SPLINE
SPL {X  -127.452, Y  +285.790, Z    +0.000, E1   +56.591, E3 +27659.937}
SPL {X  -151.591, Y  +331.344, Z    +0.000, E1   +43.870, E3 +27676.036}
SPL {X  -158.135, Y  +358.205, Z    +0.000, E1   +26.984, E3 +27679.764}
SPL {X  -159.602, Y  +371.361, Z    +0.000, E1   +14.835, E3 +27680.660}
SPL {X  -159.981, Y  +380.818, Z    +0.000, E1    +4.512, E3 +27680.938}
SPL {X  -159.990, Y  +384.681, Z    +0.000, E1    -0.222, E3 +27680.967}
SPL {X  -159.990, Y  +387.626, Z    +0.000, E1    -8.190, E3 +27680.995}
SPL {X  -159.990, Y  +390.340, Z    +0.000, E1   -15.987, E3 +27681.060}
SPL {X  -159.990, Y  +394.216, Z    +0.000, E1   -27.062, E3 +27681.222}
SPL {X  -159.990, Y  +399.855, Z    +0.000, E1   -40.916, E3 +27681.593}
SPL {X  -159.990, Y  +405.475, Z    +0.000, E1   -51.039, E3 +27682.110}
SPL {X  -159.990, Y  +414.231, Z    +0.000, E1   -60.575, E3 +27683.294}
SPL {X  -159.990, Y  +462.953, Z    +0.000, E1   -73.611, E3 +27695.033}
SPL {X  -153.839, Y  +715.436, Z    +0.000, E1   -75.884, E3 +27797.463}
SPL {X  -148.840, Y  +730.182, Z    +0.000, E1   -75.434, E3 +27810.040}
SPL {X  -143.409, Y  +742.426, Z    +0.000, E1   -74.905, E3 +27821.552}
SPL {X  -139.557, Y  +749.735, Z    +0.000, E1   -74.483, E3 +27828.900}
SPL {X  -136.371, Y  +755.165, Z    +0.000, E1   -74.152, E3 +27834.446}
SPL {X  -133.102, Y  +760.274, Z    +0.000, E1   -73.777, E3 +27839.831}
SPL {X  -128.975, Y  +766.169, Z    +0.000, E1   -73.313, E3 +27846.106}
SPL {X  -124.947, Y  +771.425, Z    +0.000, E1   -72.782, E3 +27851.799}
SPL {X  -121.698, Y  +775.357, Z    +0.000, E1   -72.353, E3 +27855.994}
SPL {X  -118.622, Y  +778.858, Z    +0.000, E1   -71.924, E3 +27859.620}
SPL {X   -66.171, Y  +817.165, Z    +0.000, E1   -56.016, E3 +28010.978}
ENDSPLINE

SPLINE
SPL {X  -126.418, Y  +769.557, Z    +0.000, E1   -57.118, E3 +28194.219}
SPL {X  -148.476, Y  +731.097, Z    +0.000, E1   -47.824, E3 +28209.375}
SPL {X  -156.642, Y  +704.059, Z    +0.000, E1   -33.659, E3 +28214.017}
SPL {X  -159.317, Y  +686.157, Z    +0.000, E1   -18.660, E3 +28215.507}
SPL {X  -159.973, Y  +673.799, Z    +0.000, E1    -5.345, E3 +28215.956}
SPL {X  -159.990, Y  +669.500, Z    +0.000, E1    +0.000, E3 +28215.996}
SPL {X  -159.990, Y  +667.794, Z    +0.000, E1    +4.255, E3 +28216.007}
SPL {X  -159.990, Y  +664.091, Z    +0.000, E1   +14.928, E3 +28216.079}
SPL {X  -159.990, Y  +659.599, Z    +0.000, E1   +28.016, E3 +28216.250}
SPL {X  -159.990, Y  +652.711, Z    +0.000, E1   +44.293, E3 +28216.729}
SPL {X  -159.990, Y  +640.730, Z    +0.000, E1   +60.297, E3 +28218.078}
SPL {X  -159.990, Y  +620.478, Z    +0.000, E1   +70.026, E3 +28221.891}
SPL {X  -159.990, Y  +573.021, Z    +0.000, E1   +74.619, E3 +28235.835}
SPL {X  -154.165, Y  +339.724, Z    +0.000, E1   +75.927, E3 +28331.682}
SPL {X  -150.223, Y  +327.456, Z    +0.000, E1   +75.573, E3 +28341.947}
SPL {X  -136.549, Y  +299.126, Z    +0.000, E1   +77.537, E3 +28334.837}
ENDSPLINE

SPLINE
SPL {X  -136.862, Y  +299.641, Z    +0.000, E1   +76.604, E3 +28343.479}
ENDSPLINE

SPLINE
SPL {X  -136.434, Y  +298.938, Z    +0.000, E1   +75.982, E3 +28349.370}
SPL {X  -135.890, Y  +298.057, Z    +0.000, E1   +75.040, E3 +28357.836}
SPL {X  -134.349, Y  +295.626, Z    +0.000, E1   +74.322, E3 +28364.683}
SPL {X  -131.287, Y  +291.064, Z    +0.000, E1   +73.972, E3 +28369.496}
SPL {X  -128.265, Y  +286.871, Z    +0.000, E1   +73.613, E3 +28373.952}
SPL {X  -125.161, Y  +282.843, Z    +0.000, E1   +73.232, E3 +28378.224}
SPL {X  -122.038, Y  +279.042, Z    +0.000, E1   +72.832, E3 +28382.204}
SPL {X  -118.642, Y  +275.165, Z    +0.000, E1   +72.381, E3 +28386.167}
SPL {X   -66.040, Y  +236.776, Z    +0.000, E1   +55.694, E3 +28547.530}
ENDSPLINE

SPLINE
SPL {X  -127.452, Y  +285.790, Z    +0.000, E1   +56.591, E3 +28721.476}
SPL {X  -151.591, Y  +331.344, Z    +0.000, E1   +43.870, E3 +28737.575}
SPL {X  -158.135, Y  +358.205, Z    +0.000, E1   +26.984, E3 +28741.302}
SPL {X  -159.602, Y  +371.361, Z    +0.000, E1   +14.835, E3 +28742.198}
SPL {X  -159.981, Y  +380.818, Z    +0.000, E1    +4.512, E3 +28742.476}
SPL {X  -159.990, Y  +384.681, Z    +0.000, E1    -0.222, E3 +28742.505}
SPL {X  -159.990, Y  +387.626, Z    +0.000, E1    -8.190, E3 +28742.534}
SPL {X  -159.990, Y  +390.340, Z    +0.000, E1   -15.987, E3 +28742.598}
SPL {X  -159.990, Y  +394.216, Z    +0.000, E1   -27.062, E3 +28742.760}
SPL {X  -159.990, Y  +399.855, Z    +0.000, E1   -40.916, E3 +28743.131}
SPL {X  -159.990, Y  +405.475, Z    +0.000, E1   -51.039, E3 +28743.648}
SPL {X  -159.990, Y  +414.231, Z    +0.000, E1   -60.575, E3 +28744.832}
SPL {X  -159.990, Y  +462.953, Z    +0.000, E1   -73.611, E3 +28756.571}
SPL {X  -153.839, Y  +715.436, Z    +0.000, E1   -75.884, E3 +28859.002}
SPL {X  -148.840, Y  +730.182, Z    +0.000, E1   -75.434, E3 +28871.578}
SPL {X  -143.409, Y  +742.426, Z    +0.000, E1   -74.905, E3 +28883.090}
SPL {X  -139.557, Y  +749.735, Z    +0.000, E1   -74.483, E3 +28890.439}
SPL {X  -136.371, Y  +755.165, Z    +0.000, E1   -74.152, E3 +28895.984}
SPL {X  -133.102, Y  +760.274, Z    +0.000, E1   -73.777, E3 +28901.369}
SPL {X  -128.975, Y  +766.169, Z    +0.000, E1   -73.313, E3 +28907.645}
SPL {X  -124.947, Y  +771.425, Z    +0.000, E1   -72.782, E3 +28913.338}
SPL {X  -121.698, Y  +775.357, Z    +0.000, E1   -72.353, E3 +28917.532}
SPL {X  -118.622, Y  +778.858, Z    +0.000, E1   -71.924, E3 +28921.158}
SPL {X   -66.171, Y  +817.165, Z    +0.000, E1   -56.016, E3 +29072.517}
ENDSPLINE

SPLINE
SPL {X  -126.418, Y  +769.557, Z    +0.000, E1   -57.118, E3 +29255.758}
SPL {X  -148.476, Y  +731.097, Z    +0.000, E1   -47.824, E3 +29270.914}
SPL {X  -156.642, Y  +704.059, Z    +0.000, E1   -33.659, E3 +29275.555}
SPL {X  -159.317, Y  +686.157, Z    +0.000, E1   -18.660, E3 +29277.046}
SPL {X  -159.973, Y  +673.799, Z    +0.000, E1    -5.345, E3 +29277.494}
SPL {X  -159.990, Y  +669.500, Z    +0.000, E1    +0.000, E3 +29277.534}
SPL {X  -159.990, Y  +667.794, Z    +0.000, E1    +4.255, E3 +29277.546}
SPL {X  -159.990, Y  +664.091, Z    +0.000, E1   +14.928, E3 +29277.618}
SPL {X  -159.990, Y  +659.599, Z    +0.000, E1   +28.016, E3 +29277.788}
SPL {X  -159.990, Y  +652.711, Z    +0.000, E1   +44.293, E3 +29278.268}
SPL {X  -159.990, Y  +640.730, Z    +0.000, E1   +60.297, E3 +29279.617}
SPL {X  -159.990, Y  +620.478, Z    +0.000, E1   +70.026, E3 +29283.430}
SPL {X  -159.990, Y  +573.021, Z    +0.000, E1   +74.619, E3 +29297.374}
SPL {X  -154.165, Y  +339.724, Z    +0.000, E1   +75.927, E3 +29393.221}
SPL {X  -150.223, Y  +327.456, Z    +0.000, E1   +75.573, E3 +29403.486}
SPL {X  -136.549, Y  +299.126, Z    +0.000, E1   +77.537, E3 +29396.376}
ENDSPLINE

SPLINE
SPL {X  -136.862, Y  +299.641, Z    +0.000, E1   +76.604, E3 +29405.018}
ENDSPLINE

SPLINE
SPL {X  -136.434, Y  +298.938, Z    +0.000, E1   +75.982, E3 +29410.909}
SPL {X  -135.890, Y  +298.057, Z    +0.000, E1   +75.040, E3 +29419.375}
SPL {X  -134.349, Y  +295.626, Z    +0.000, E1   +74.322, E3 +29426.222}
SPL {X  -131.287, Y  +291.064, Z    +0.000, E1   +73.972, E3 +29431.034}
SPL {X  -128.265, Y  +286.871, Z    +0.000, E1   +73.613, E3 +29435.490}
SPL {X  -125.161, Y  +282.843, Z    +0.000, E1   +73.232, E3 +29439.762}
SPL {X  -122.038, Y  +279.042, Z    +0.000, E1   +72.832, E3 +29443.742}
SPL {X  -118.642, Y  +275.165, Z    +0.000, E1   +72.381, E3 +29447.705}
SPL {X   -66.040, Y  +236.776, Z    +0.000, E1   +55.694, E3 +29609.069}
ENDSPLINE

SPLINE
SPL {X  -127.452, Y  +285.790, Z    +0.000, E1   +56.591, E3 +29783.014}
SPL {X  -151.591, Y  +331.344, Z    +0.000, E1   +43.870, E3 +29799.113}
SPL {X  -158.135, Y  +358.205, Z    +0.000, E1   +26.984, E3 +29802.841}
SPL {X  -159.602, Y  +371.361, Z    +0.000, E1   +14.835, E3 +29803.737}
SPL {X  -159.981, Y  +380.818, Z    +0.000, E1    +4.512, E3 +29804.015}
SPL {X  -159.990, Y  +384.681, Z    +0.000, E1    -0.222, E3 +29804.044}
SPL {X  -159.990, Y  +387.626, Z    +0.000, E1    -8.190, E3 +29804.072}
SPL {X  -159.990, Y  +390.340, Z    +0.000, E1   -15.987, E3 +29804.137}
SPL {X  -159.990, Y  +394.216, Z    +0.000, E1   -27.062, E3 +29804.299}
SPL {X  -159.990, Y  +399.855, Z    +0.000, E1   -40.916, E3 +29804.670}
SPL {X  -159.990, Y  +405.475, Z    +0.000, E1   -51.039, E3 +29805.187}
SPL {X  -159.990, Y  +414.231, Z    +0.000, E1   -60.575, E3 +29806.371}
SPL {X  -159.990, Y  +462.953, Z    +0.000, E1   -73.611, E3 +29818.110}
SPL {X  -153.839, Y  +715.436, Z    +0.000, E1   -75.884, E3 +29920.540}
SPL {X  -149.923, Y  +727.355, Z    +0.000, E1   -75.515, E3 +29930.650}
SPL {X  -145.995, Y  +736.939, Z    +0.000, E1   -75.150, E3 +29939.385}
SPL {X  -141.012, Y  +747.080, Z    +0.000, E1   -74.661, E3 +29949.237}
SPL {X  -136.371, Y  +755.165, Z    +0.000, E1   -74.152, E3 +29957.523}
SPL {X  -133.102, Y  +760.274, Z    +0.000, E1   -73.777, E3 +29962.908}
SPL {X  -128.975, Y  +766.169, Z    +0.000, E1   -73.313, E3 +29969.183}
SPL {X  -124.947, Y  +771.425, Z    +0.000, E1   -72.782, E3 +29974.876}
SPL {X  -121.698, Y  +775.357, Z    +0.000, E1   -72.353, E3 +29979.071}
SPL {X  -118.622, Y  +778.858, Z    +0.000, E1   -71.924, E3 +29982.697}
SPL {X   -66.171, Y  +817.165, Z    +0.000, E1   -56.016, E3 +30134.055}
ENDSPLINE

SPLINE
SPL {X  -126.418, Y  +769.557, Z    +0.000, E1   -57.118, E3 +30317.296}
SPL {X  -148.476, Y  +731.097, Z    +0.000, E1   -47.824, E3 +30332.452}
SPL {X  -156.642, Y  +704.059, Z    +0.000, E1   -33.659, E3 +30337.094}
SPL {X  -159.317, Y  +686.157, Z    +0.000, E1   -18.660, E3 +30338.584}
SPL {X  -159.907, Y  +676.666, Z    +0.000, E1    -8.555, E3 +30338.982}
SPL {X  -159.990, Y  +669.586, Z    +0.000, E1    -0.216, E3 +30339.073}
SPL {X  -159.990, Y  +667.794, Z    +0.000, E1    +4.255, E3 +30339.084}
SPL {X  -159.990, Y  +664.091, Z    +0.000, E1   +14.928, E3 +30339.156}
SPL {X  -159.990, Y  +659.599, Z    +0.000, E1   +28.016, E3 +30339.327}
SPL {X  -159.990, Y  +652.711, Z    +0.000, E1   +44.293, E3 +30339.806}
SPL {X  -159.990, Y  +640.730, Z    +0.000, E1   +60.297, E3 +30341.155}
SPL {X  -159.990, Y  +620.478, Z    +0.000, E1   +70.026, E3 +30344.968}
SPL {X  -159.990, Y  +573.021, Z    +0.000, E1   +74.619, E3 +30358.912}
SPL {X  -154.165, Y  +339.724, Z    +0.000, E1   +75.927, E3 +30454.759}
SPL {X  -150.223, Y  +327.456, Z    +0.000, E1   +75.573, E3 +30465.024}
SPL {X  -136.549, Y  +299.126, Z    +0.000, E1   +77.537, E3 +30457.914}
ENDSPLINE

SPLINE
SPL {X  -136.862, Y  +299.641, Z    +0.000, E1   +76.604, E3 +30466.556}
ENDSPLINE

SPLINE
SPL {X  -136.434, Y  +298.938, Z    +0.000, E1   +75.982, E3 +30472.447}
SPL {X  -135.890, Y  +298.057, Z    +0.000, E1   +75.040, E3 +30480.913}
SPL {X  -134.349, Y  +295.626, Z    +0.000, E1   +74.322, E3 +30487.760}
SPL {X  -131.287, Y  +291.064, Z    +0.000, E1   +73.972, E3 +30492.573}
SPL {X  -128.265, Y  +286.871, Z    +0.000, E1   +73.613, E3 +30497.029}
SPL {X  -125.161, Y  +282.843, Z    +0.000, E1   +73.232, E3 +30501.301}
SPL {X  -122.038, Y  +279.042, Z    +0.000, E1   +72.832, E3 +30505.281}
SPL {X  -118.642, Y  +275.165, Z    +0.000, E1   +72.381, E3 +30509.244}
SPL {X   -66.040, Y  +236.776, Z    +0.000, E1   +55.694, E3 +30670.607}
ENDSPLINE

SPLINE
SPL {X  -127.452, Y  +285.790, Z    +0.000, E1   +56.591, E3 +30844.552}
SPL {X  -148.001, Y  +321.733, Z    +0.000, E1   +47.810, E3 +30858.656}
SPL {X  -154.604, Y  +341.337, Z    +0.000, E1   +38.630, E3 +30862.430}
SPL {X  -158.135, Y  +358.205, Z    +0.000, E1   +26.984, E3 +30864.379}
SPL {X  -159.602, Y  +371.361, Z    +0.000, E1   +14.835, E3 +30865.275}
SPL {X  -159.981, Y  +380.818, Z    +0.000, E1    +4.512, E3 +30865.553}
SPL {X  -159.990, Y  +384.681, Z    +0.000, E1    -0.222, E3 +30865.582}
SPL {X  -159.990, Y  +389.079, Z    +0.000, E1   -12.017, E3 +30865.645}
SPL {X  -159.990, Y  +394.216, Z    +0.000, E1   -27.062, E3 +30865.837}
SPL {X  -159.990, Y  +399.855, Z    +0.000, E1   -40.916, E3 +30866.208}
SPL {X  -159.990, Y  +405.475, Z    +0.000, E1   -51.039, E3 +30866.725}
SPL {X  -159.990, Y  +414.231, Z    +0.000, E1   -60.575, E3 +30867.909}
SPL {X  -159.990, Y  +462.953, Z    +0.000, E1   -73.611, E3 +30879.648}
SPL {X  -153.839, Y  +715.436, Z    +0.000, E1   -75.884, E3 +30982.079}
SPL {X  -148.840, Y  +730.182, Z    +0.000, E1   -75.434, E3 +30994.655}
SPL {X  -143.409, Y  +742.426, Z    +0.000, E1   -74.905, E3 +31006.167}
SPL {X  -139.557, Y  +749.735, Z    +0.000, E1   -74.483, E3 +31013.515}
SPL {X  -136.371, Y  +755.165, Z    +0.000, E1   -74.152, E3 +31019.061}
SPL {X  -133.102, Y  +760.274, Z    +0.000, E1   -73.777, E3 +31024.446}
SPL {X  -128.975, Y  +766.169, Z    +0.000, E1   -73.313, E3 +31030.722}
SPL {X  -124.947, Y  +771.425, Z    +0.000, E1   -72.782, E3 +31036.415}
SPL {X  -121.698, Y  +775.357, Z    +0.000, E1   -72.353, E3 +31040.609}
SPL {X  -118.622, Y  +778.858, Z    +0.000, E1   -71.924, E3 +31044.235}
SPL {X   -66.171, Y  +817.165, Z    +0.000, E1   -56.016, E3 +31195.593}
ENDSPLINE

SPLINE
SPL {X  -126.418, Y  +769.557, Z    +0.000, E1   -57.118, E3 +31378.835}
SPL {X  -145.244, Y  +738.589, Z    +0.000, E1   -50.405, E3 +31392.076}
SPL {X  -150.151, Y  +726.741, Z    +0.000, E1   -46.068, E3 +31395.003}
SPL {X  -156.642, Y  +704.059, Z    +0.000, E1   -33.659, E3 +31398.632}
SPL {X  -159.317, Y  +686.157, Z    +0.000, E1   -18.660, E3 +31400.123}
SPL {X  -159.973, Y  +673.799, Z    +0.000, E1    -5.345, E3 +31400.571}
SPL {X  -159.990, Y  +669.500, Z    +0.000, E1    +0.000, E3 +31400.611}
SPL {X  -159.990, Y  +667.794, Z    +0.000, E1    +4.255, E3 +31400.623}
SPL {X  -159.990, Y  +664.091, Z    +0.000, E1   +14.928, E3 +31400.695}
SPL {X  -159.990, Y  +658.301, Z    +0.000, E1   +31.283, E3 +31400.947}
SPL {X  -159.990, Y  +650.845, Z    +0.000, E1   +47.892, E3 +31401.492}
SPL {X  -159.990, Y  +640.730, Z    +0.000, E1   +60.297, E3 +31402.693}
SPL {X  -159.990, Y  +620.478, Z    +0.000, E1   +70.026, E3 +31406.507}
SPL {X  -159.990, Y  +573.021, Z    +0.000, E1   +74.619, E3 +31420.451}
SPL {X  -154.165, Y  +339.724, Z    +0.000, E1   +75.927, E3 +31516.298}
SPL {X  -150.223, Y  +327.456, Z    +0.000, E1   +75.573, E3 +31526.562}
SPL {X  -136.549, Y  +299.126, Z    +0.000, E1   +77.537, E3 +31519.452}
ENDSPLINE

SPLINE
SPL {X  -136.862, Y  +299.641, Z    +0.000, E1   +76.604, E3 +31528.094}
ENDSPLINE

SPLINE
SPL {X  -136.434, Y  +298.938, Z    +0.000, E1   +75.982, E3 +31533.986}
SPL {X  -135.890, Y  +298.057, Z    +0.000, E1   +75.040, E3 +31542.452}
SPL {X  -134.349, Y  +295.626, Z    +0.000, E1   +74.322, E3 +31549.299}
SPL {X  -131.287, Y  +291.064, Z    +0.000, E1   +73.972, E3 +31554.111}
SPL {X  -128.265, Y  +286.871, Z    +0.000, E1   +73.613, E3 +31558.567}
SPL {X  -125.161, Y  +282.843, Z    +0.000, E1   +73.232, E3 +31562.839}
SPL {X  -122.038, Y  +279.042, Z    +0.000, E1   +72.832, E3 +31566.819}
SPL {X  -118.642, Y  +275.165, Z    +0.000, E1   +72.381, E3 +31570.782}
SPL {X   -66.040, Y  +236.776, Z    +0.000, E1   +55.694, E3 +31732.146}
ENDSPLINE

SPLINE
SPL {X  -127.452, Y  +285.790, Z    +0.000, E1   +56.591, E3 +31906.091}
SPL {X  -151.591, Y  +331.344, Z    +0.000, E1   +43.870, E3 +31922.190}
SPL {X  -158.135, Y  +358.205, Z    +0.000, E1   +26.984, E3 +31925.918}
SPL {X  -159.602, Y  +371.361, Z    +0.000, E1   +14.835, E3 +31926.814}
SPL {X  -159.981, Y  +380.818, Z    +0.000, E1    +4.512, E3 +31927.092}
SPL {X  -159.990, Y  +384.681, Z    +0.000, E1    -0.222, E3 +31927.121}
SPL {X  -159.990, Y  +387.626, Z    +0.000, E1    -8.190, E3 +31927.149}
SPL {X  -159.990, Y  +390.340, Z    +0.000, E1   -15.987, E3 +31927.214}
SPL {X  -159.990, Y  +394.216, Z    +0.000, E1   -27.062, E3 +31927.375}
SPL {X  -159.990, Y  +399.855, Z    +0.000, E1   -40.916, E3 +31927.747}
SPL {X  -159.990, Y  +405.475, Z    +0.000, E1   -51.039, E3 +31928.263}
SPL {X  -159.990, Y  +414.231, Z    +0.000, E1   -60.575, E3 +31929.448}
SPL {X  -159.990, Y  +462.953, Z    +0.000, E1   -73.611, E3 +31941.187}
SPL {X  -153.839, Y  +715.436, Z    +0.000, E1   -75.884, E3 +32043.617}
SPL {X  -149.923, Y  +727.355, Z    +0.000, E1   -75.515, E3 +32053.727}
SPL {X  -145.995, Y  +736.939, Z    +0.000, E1   -75.150, E3 +32062.462}
SPL {X  -141.012, Y  +747.080, Z    +0.000, E1   -74.661, E3 +32072.314}
SPL {X  -136.371, Y  +755.165, Z    +0.000, E1   -74.152, E3 +32080.600}
SPL {X  -131.455, Y  +762.694, Z    +0.000, E1   -73.615, E3 +32088.518}
SPL {X  -125.933, Y  +770.180, Z    +0.000, E1   -72.934, E3 +32096.582}
SPL {X  -121.698, Y  +775.357, Z    +0.000, E1   -72.353, E3 +32102.148}
SPL {X  -118.622, Y  +778.858, Z    +0.000, E1   -71.924, E3 +32105.774}
SPL {X   -66.171, Y  +817.165, Z    +0.000, E1   -56.016, E3 +32257.132}
ENDSPLINE

SPLINE
SPL {X  -126.418, Y  +769.557, Z    +0.000, E1   -57.118, E3 +32440.373}
SPL {X  -145.244, Y  +738.589, Z    +0.000, E1   -50.405, E3 +32453.615}
SPL {X  -150.151, Y  +726.741, Z    +0.000, E1   -46.068, E3 +32456.541}
SPL {X  -156.642, Y  +704.059, Z    +0.000, E1   -33.659, E3 +32460.171}
SPL {X  -159.317, Y  +686.157, Z    +0.000, E1   -18.660, E3 +32461.661}
SPL {X  -159.973, Y  +673.799, Z    +0.000, E1    -5.345, E3 +32462.110}
SPL {X  -159.990, Y  +669.500, Z    +0.000, E1    +0.000, E3 +32462.150}
SPL {X  -159.990, Y  +667.794, Z    +0.000, E1    +4.255, E3 +32462.161}
SPL {X  -159.990, Y  +664.091, Z    +0.000, E1   +14.928, E3 +32462.233}
SPL {X  -159.990, Y  +658.301, Z    +0.000, E1   +31.283, E3 +32462.486}
SPL {X  -159.990, Y  +650.845, Z    +0.000, E1   +47.892, E3 +32463.031}
SPL {X  -159.990, Y  +640.730, Z    +0.000, E1   +60.297, E3 +32464.232}
SPL {X  -159.990, Y  +620.478, Z    +0.000, E1   +70.026, E3 +32468.045}
SPL {X  -159.990, Y  +573.021, Z    +0.000, E1   +74.619, E3 +32481.989}
SPL {X  -154.165, Y  +339.724, Z    +0.000, E1   +75.927, E3 +32577.836}
SPL {X  -150.223, Y  +327.456, Z    +0.000, E1   +75.573, E3 +32588.101}
SPL {X  -136.549, Y  +299.126, Z    +0.000, E1   +77.537, E3 +32580.991}
ENDSPLINE

SPLINE
SPL {X  -136.862, Y  +299.641, Z    +0.000, E1   +76.604, E3 +32589.633}
ENDSPLINE

SPLINE
SPL {X  -136.434, Y  +298.938, Z    +0.000, E1   +75.982, E3 +32595.524}
SPL {X  -135.890, Y  +298.057, Z    +0.000, E1   +75.040, E3 +32603.990}
SPL {X  -134.349, Y  +295.626, Z    +0.000, E1   +74.322, E3 +32610.837}
SPL {X  -131.287, Y  +291.064, Z    +0.000, E1   +73.972, E3 +32615.650}
SPL {X  -128.265, Y  +286.871, Z    +0.000, E1   +73.613, E3 +32620.106}
SPL {X  -125.161, Y  +282.843, Z    +0.000, E1   +73.232, E3 +32624.378}
SPL {X  -122.038, Y  +279.042, Z    +0.000, E1   +72.832, E3 +32628.357}
SPL {X  -118.642, Y  +275.165, Z    +0.000, E1   +72.381, E3 +32632.321}
SPL {X   -66.040, Y  +236.776, Z    +0.000, E1   +55.694, E3 +32793.684}
ENDSPLINE

SPLINE
SPL {X  -127.452, Y  +285.790, Z    +0.000, E1   +56.591, E3 +32967.629}
SPL {X  -151.591, Y  +331.344, Z    +0.000, E1   +43.870, E3 +32983.729}
SPL {X  -158.135, Y  +358.205, Z    +0.000, E1   +26.984, E3 +32987.456}
SPL {X  -159.602, Y  +371.361, Z    +0.000, E1   +14.835, E3 +32988.352}
SPL {X  -159.981, Y  +380.818, Z    +0.000, E1    +4.512, E3 +32988.630}
SPL {X  -159.990, Y  +384.681, Z    +0.000, E1    -0.222, E3 +32988.659}
SPL {X  -159.990, Y  +387.626, Z    +0.000, E1    -8.190, E3 +32988.687}
SPL {X  -159.990, Y  +390.340, Z    +0.000, E1   -15.987, E3 +32988.752}
SPL {X  -159.990, Y  +394.216, Z    +0.000, E1   -27.062, E3 +32988.914}
SPL {X  -159.990, Y  +399.855, Z    +0.000, E1   -40.916, E3 +32989.285}
SPL {X  -159.990, Y  +405.475, Z    +0.000, E1   -51.039, E3 +32989.802}
SPL {X  -159.990, Y  +414.231, Z    +0.000, E1   -60.575, E3 +32990.986}
SPL {X  -159.990, Y  +462.953, Z    +0.000, E1   -73.611, E3 +33002.725}
SPL {X  -153.839, Y  +715.436, Z    +0.000, E1   -75.884, E3 +33105.156}
SPL {X  -148.840, Y  +730.182, Z    +0.000, E1   -75.434, E3 +33117.732}
SPL {X  -143.409, Y  +742.426, Z    +0.000, E1   -74.905, E3 +33129.244}
SPL {X  -139.557, Y  +749.735, Z    +0.000, E1   -74.483, E3 +33136.592}
SPL {X  -136.371, Y  +755.165, Z    +0.000, E1   -74.152, E3 +33142.138}
SPL {X  -133.102, Y  +760.274, Z    +0.000, E1   -73.777, E3 +33147.523}
SPL {X  -128.975, Y  +766.169, Z    +0.000, E1   -73.313, E3 +33153.799}
SPL {X  -124.947, Y  +771.425, Z    +0.000, E1   -72.782, E3 +33159.492}
SPL {X  -121.698, Y  +775.357, Z    +0.000, E1   -72.353, E3 +33163.686}
SPL {X  -118.622, Y  +778.858, Z    +0.000, E1   -71.924, E3 +33167.312}
SPL {X   -66.171, Y  +817.165, Z    +0.000, E1   -56.016, E3 +33318.670}
ENDSPLINE

SPLINE
SPL {X  -126.418, Y  +769.557, Z    +0.000, E1   -57.118, E3 +33501.912}
SPL {X  -145.244, Y  +738.589, Z    +0.000, E1   -50.405, E3 +33515.153}
SPL {X  -150.151, Y  +726.741, Z    +0.000, E1   -46.068, E3 +33518.080}
SPL {X  -156.642, Y  +704.059, Z    +0.000, E1   -33.659, E3 +33521.709}
SPL {X  -159.317, Y  +686.157, Z    +0.000, E1   -18.660, E3 +33523.200}
SPL {X  -159.973, Y  +673.799, Z    +0.000, E1    -5.345, E3 +33523.648}
SPL {X  -159.990, Y  +669.500, Z    +0.000, E1    +0.000, E3 +33523.688}
SPL {X  -159.990, Y  +667.794, Z    +0.000, E1    +4.255, E3 +33523.699}
SPL {X  -159.990, Y  +664.091, Z    +0.000, E1   +14.928, E3 +33523.772}
SPL {X  -159.990, Y  +659.599, Z    +0.000, E1   +28.016, E3 +33523.942}
SPL {X  -159.990, Y  +652.711, Z    +0.000, E1   +44.293, E3 +33524.421}
SPL {X  -159.990, Y  +640.730, Z    +0.000, E1   +60.297, E3 +33525.770}
SPL {X  -159.990, Y  +620.478, Z    +0.000, E1   +70.026, E3 +33529.584}
SPL {X  -159.990, Y  +573.021, Z    +0.000, E1   +74.619, E3 +33543.528}
SPL {X  -154.165, Y  +339.724, Z    +0.000, E1   +75.927, E3 +33639.374}
SPL {X  -150.571, Y  +328.416, Z    +0.000, E1   +75.599, E3 +33648.820}
SPL {X  -148.206, Y  +322.236, Z    +0.000, E1   +75.365, E3 +33654.364}
SPL {X  -136.549, Y  +299.126, Z    +0.000, E1   +77.537, E3 +33642.529}
ENDSPLINE

SPLINE
SPL {X  -136.862, Y  +299.641, Z    +0.000, E1   +76.604, E3 +33651.171}
ENDSPLINE

SPLINE
SPL {X  -136.434, Y  +298.938, Z    +0.000, E1   +75.982, E3 +33657.062}
SPL {X  -135.890, Y  +298.057, Z    +0.000, E1   +75.040, E3 +33665.528}
SPL {X  -134.349, Y  +295.626, Z    +0.000, E1   +74.322, E3 +33672.376}
SPL {X  -131.287, Y  +291.064, Z    +0.000, E1   +73.972, E3 +33677.188}
SPL {X  -128.265, Y  +286.871, Z    +0.000, E1   +73.613, E3 +33681.644}
SPL {X  -125.161, Y  +282.843, Z    +0.000, E1   +73.232, E3 +33685.916}
SPL {X  -122.038, Y  +279.042, Z    +0.000, E1   +72.832, E3 +33689.896}
SPL {X  -118.642, Y  +275.165, Z    +0.000, E1   +72.381, E3 +33693.859}
SPL {X   -66.040, Y  +236.776, Z    +0.000, E1   +55.694, E3 +33855.223}
ENDSPLINE

SPLINE
SPL {X  -127.452, Y  +285.790, Z    +0.000, E1   +56.591, E3 +34029.168}
SPL {X  -151.591, Y  +331.344, Z    +0.000, E1   +43.870, E3 +34045.267}
SPL {X  -158.135, Y  +358.205, Z    +0.000, E1   +26.984, E3 +34048.995}
SPL {X  -159.602, Y  +371.361, Z    +0.000, E1   +14.835, E3 +34049.891}
SPL {X  -159.981, Y  +380.818, Z    +0.000, E1    +4.512, E3 +34050.169}
SPL {X  -159.990, Y  +384.681, Z    +0.000, E1    -0.222, E3 +34050.198}
SPL {X  -159.990, Y  +387.626, Z    +0.000, E1    -8.190, E3 +34050.226}
SPL {X  -159.990, Y  +390.340, Z    +0.000, E1   -15.987, E3 +34050.290}
SPL {X  -159.990, Y  +394.216, Z    +0.000, E1   -27.062, E3 +34050.452}
SPL {X  -159.990, Y  +399.855, Z    +0.000, E1   -40.916, E3 +34050.823}
SPL {X  -159.990, Y  +405.475, Z    +0.000, E1   -51.039, E3 +34051.340}
SPL {X  -159.990, Y  +414.231, Z    +0.000, E1   -60.575, E3 +34052.525}
SPL {X  -159.990, Y  +462.953, Z    +0.000, E1   -73.611, E3 +34064.264}
SPL {X  -153.839, Y  +715.436, Z    +0.000, E1   -75.884, E3 +34166.694}
SPL {X  -148.840, Y  +730.182, Z    +0.000, E1   -75.434, E3 +34179.271}
SPL {X  -143.409, Y  +742.426, Z    +0.000, E1   -74.905, E3 +34190.783}
SPL {X  -139.557, Y  +749.735, Z    +0.000, E1   -74.483, E3 +34198.131}
SPL {X  -136.371, Y  +755.165, Z    +0.000, E1   -74.152, E3 +34203.677}
SPL {X  -133.102, Y  +760.274, Z    +0.000, E1   -73.777, E3 +34209.062}
SPL {X  -128.975, Y  +766.169, Z    +0.000, E1   -73.313, E3 +34215.337}
SPL {X  -124.947, Y  +771.425, Z    +0.000, E1   -72.782, E3 +34221.030}
SPL {X  -121.698, Y  +775.357, Z    +0.000, E1   -72.353, E3 +34225.225}
SPL {X  -118.622, Y  +778.858, Z    +0.000, E1   -71.924, E3 +34228.851}
SPL {X   -66.171, Y  +817.165, Z    +0.000, E1   -56.016, E3 +34380.209}
ENDSPLINE

SPLINE
SPL {X  -126.418, Y  +769.557, Z    +0.000, E1   -57.118, E3 +34563.450}
SPL {X  -148.476, Y  +731.097, Z    +0.000, E1   -47.824, E3 +34578.606}
SPL {X  -156.642, Y  +704.059, Z    +0.000, E1   -33.659, E3 +34583.248}
SPL {X  -159.317, Y  +686.157, Z    +0.000, E1   -18.660, E3 +34584.738}
SPL {X  -159.973, Y  +673.799, Z    +0.000, E1    -5.345, E3 +34585.187}
SPL {X  -159.990, Y  +669.500, Z    +0.000, E1    +0.000, E3 +34585.227}
SPL {X  -159.990, Y  +667.794, Z    +0.000, E1    +4.255, E3 +34585.238}
SPL {X  -159.990, Y  +664.091, Z    +0.000, E1   +14.928, E3 +34585.310}
SPL {X  -159.990, Y  +659.599, Z    +0.000, E1   +28.016, E3 +34585.480}
SPL {X  -159.990, Y  +652.711, Z    +0.000, E1   +44.293, E3 +34585.960}
SPL {X  -159.990, Y  +640.730, Z    +0.000, E1   +60.297, E3 +34587.309}
SPL {X  -159.990, Y  +620.478, Z    +0.000, E1   +70.026, E3 +34591.122}
SPL {X  -159.990, Y  +573.021, Z    +0.000, E1   +74.619, E3 +34605.066}
SPL {X  -154.165, Y  +339.724, Z    +0.000, E1   +75.927, E3 +34700.913}
SPL {X  -150.223, Y  +327.456, Z    +0.000, E1   +75.573, E3 +34711.178}
SPL {X  -136.549, Y  +299.126, Z    +0.000, E1   +77.537, E3 +34704.068}
ENDSPLINE

SPLINE
SPL {X  -136.862, Y  +299.641, Z    +0.000, E1   +76.604, E3 +34712.710}
ENDSPLINE

SPLINE
SPL {X  -136.434, Y  +298.938, Z    +0.000, E1   +75.982, E3 +34718.601}
SPL {X  -135.890, Y  +298.057, Z    +0.000, E1   +75.040, E3 +34727.067}
SPL {X  -134.349, Y  +295.626, Z    +0.000, E1   +74.322, E3 +34733.914}
SPL {X  -131.287, Y  +291.064, Z    +0.000, E1   +73.972, E3 +34738.727}
SPL {X  -128.265, Y  +286.871, Z    +0.000, E1   +73.613, E3 +34743.183}
SPL {X  -125.161, Y  +282.843, Z    +0.000, E1   +73.232, E3 +34747.454}
SPL {X  -122.038, Y  +279.042, Z    +0.000, E1   +72.832, E3 +34751.434}
SPL {X  -118.642, Y  +275.165, Z    +0.000, E1   +72.381, E3 +34755.398}
SPL {X   -66.040, Y  +236.776, Z    +0.000, E1   +55.694, E3 +34916.761}
ENDSPLINE

SPLINE
SPL {X  -127.452, Y  +285.790, Z    +0.000, E1   +56.591, E3 +35090.706}
SPL {X  -151.591, Y  +331.344, Z    +0.000, E1   +43.870, E3 +35106.806}
SPL {X  -158.135, Y  +358.205, Z    +0.000, E1   +26.984, E3 +35110.533}
SPL {X  -159.602, Y  +371.361, Z    +0.000, E1   +14.835, E3 +35111.429}
SPL {X  -159.981, Y  +380.818, Z    +0.000, E1    +4.512, E3 +35111.707}
SPL {X  -159.990, Y  +384.681, Z    +0.000, E1    -0.222, E3 +35111.736}
SPL {X  -159.990, Y  +387.626, Z    +0.000, E1    -8.190, E3 +35111.764}
SPL {X  -159.990, Y  +390.340, Z    +0.000, E1   -15.987, E3 +35111.829}
SPL {X  -159.990, Y  +394.216, Z    +0.000, E1   -27.062, E3 +35111.991}
SPL {X  -159.990, Y  +399.855, Z    +0.000, E1   -40.916, E3 +35112.362}
SPL {X  -159.990, Y  +405.475, Z    +0.000, E1   -51.039, E3 +35112.879}
SPL {X  -159.990, Y  +414.231, Z    +0.000, E1   -60.575, E3 +35114.063}
SPL {X  -159.990, Y  +462.953, Z    +0.000, E1   -73.611, E3 +35125.802}
SPL {X  -153.839, Y  +715.436, Z    +0.000, E1   -75.884, E3 +35228.233}
SPL {X  -148.840, Y  +730.182, Z    +0.000, E1   -75.434, E3 +35240.809}
SPL {X  -143.409, Y  +742.426, Z    +0.000, E1   -74.905, E3 +35252.321}
SPL {X  -139.557, Y  +749.735, Z    +0.000, E1   -74.483, E3 +35259.669}
SPL {X  -136.371, Y  +755.165, Z    +0.000, E1   -74.152, E3 +35265.215}
SPL {X  -133.102, Y  +760.274, Z    +0.000, E1   -73.777, E3 +35270.600}
SPL {X  -128.975, Y  +766.169, Z    +0.000, E1   -73.313, E3 +35276.875}
SPL {X  -124.947, Y  +771.425, Z    +0.000, E1   -72.782, E3 +35282.568}
SPL {X  -121.698, Y  +775.357, Z    +0.000, E1   -72.353, E3 +35286.763}
SPL {X  -118.622, Y  +778.858, Z    +0.000, E1   -71.924, E3 +35290.389}
SPL {X   -66.171, Y  +817.165, Z    +0.000, E1   -56.016, E3 +35441.747}
ENDSPLINE

SPLINE
SPL {X  -126.418, Y  +769.557, Z    +0.000, E1   -57.118, E3 +35624.989}
SPL {X  -148.476, Y  +731.097, Z    +0.000, E1   -47.824, E3 +35640.145}
SPL {X  -156.642, Y  +704.059, Z    +0.000, E1   -33.659, E3 +35644.786}
SPL {X  -159.317, Y  +686.157, Z    +0.000, E1   -18.660, E3 +35646.276}
SPL {X  -159.973, Y  +673.799, Z    +0.000, E1    -5.345, E3 +35646.725}
SPL {X  -159.990, Y  +669.500, Z    +0.000, E1    +0.000, E3 +35646.765}
SPL {X  -159.990, Y  +667.794, Z    +0.000, E1    +4.255, E3 +35646.776}
SPL {X  -159.990, Y  +664.091, Z    +0.000, E1   +14.928, E3 +35646.848}
SPL {X  -159.990, Y  +659.599, Z    +0.000, E1   +28.016, E3 +35647.019}
SPL {X  -159.990, Y  +652.711, Z    +0.000, E1   +44.293, E3 +35647.498}
SPL {X  -159.990, Y  +640.730, Z    +0.000, E1   +60.297, E3 +35648.847}
SPL {X  -159.990, Y  +620.478, Z    +0.000, E1   +70.026, E3 +35652.661}
SPL {X  -159.990, Y  +573.021, Z    +0.000, E1   +74.619, E3 +35666.604}
SPL {X  -154.165, Y  +339.724, Z    +0.000, E1   +75.927, E3 +35762.451}
SPL {X  -150.223, Y  +327.456, Z    +0.000, E1   +75.573, E3 +35772.716}
SPL {X  -136.549, Y  +299.126, Z    +0.000, E1   +77.537, E3 +35765.606}
ENDSPLINE

SPLINE
SPL {X  -136.862, Y  +299.641, Z    +0.000, E1   +76.604, E3 +35774.248}
ENDSPLINE

SPLINE
SPL {X  -136.434, Y  +298.938, Z    +0.000, E1   +75.982, E3 +35780.139}
SPL {X  -135.890, Y  +298.057, Z    +0.000, E1   +75.040, E3 +35788.605}
SPL {X  -134.349, Y  +295.626, Z    +0.000, E1   +74.322, E3 +35795.453}
SPL {X  -131.287, Y  +291.064, Z    +0.000, E1   +73.972, E3 +35800.265}
SPL {X  -128.265, Y  +286.871, Z    +0.000, E1   +73.613, E3 +35804.721}
SPL {X  -125.161, Y  +282.843, Z    +0.000, E1   +73.232, E3 +35808.993}
SPL {X  -122.038, Y  +279.042, Z    +0.000, E1   +72.832, E3 +35812.973}
SPL {X  -118.642, Y  +275.165, Z    +0.000, E1   +72.381, E3 +35816.936}
SPL {X   -66.040, Y  +236.776, Z    +0.000, E1   +55.694, E3 +35978.299}
ENDSPLINE

SPLINE
SPL {X  -127.452, Y  +285.790, Z    +0.000, E1   +56.591, E3 +36152.245}
SPL {X  -151.591, Y  +331.344, Z    +0.000, E1   +43.870, E3 +36168.344}
SPL {X  -158.135, Y  +358.205, Z    +0.000, E1   +26.984, E3 +36172.072}
SPL {X  -159.602, Y  +371.361, Z    +0.000, E1   +14.835, E3 +36172.968}
SPL {X  -159.981, Y  +380.818, Z    +0.000, E1    +4.512, E3 +36173.246}
SPL {X  -159.990, Y  +384.681, Z    +0.000, E1    -0.222, E3 +36173.274}
SPL {X  -159.990, Y  +387.626, Z    +0.000, E1    -8.190, E3 +36173.303}
SPL {X  -159.990, Y  +390.340, Z    +0.000, E1   -15.987, E3 +36173.367}
SPL {X  -159.990, Y  +394.216, Z    +0.000, E1   -27.062, E3 +36173.529}
SPL {X  -159.990, Y  +399.855, Z    +0.000, E1   -40.916, E3 +36173.900}
SPL {X  -159.990, Y  +405.475, Z    +0.000, E1   -51.039, E3 +36174.417}
SPL {X  -159.990, Y  +414.231, Z    +0.000, E1   -60.575, E3 +36175.602}
SPL {X  -159.990, Y  +462.953, Z    +0.000, E1   -73.611, E3 +36187.341}
SPL {X  -153.839, Y  +715.436, Z    +0.000, E1   -75.884, E3 +36289.771}
SPL {X  -148.840, Y  +730.182, Z    +0.000, E1   -75.434, E3 +36302.348}
SPL {X  -143.409, Y  +742.426, Z    +0.000, E1   -74.905, E3 +36313.860}
SPL {X  -139.557, Y  +749.735, Z    +0.000, E1   -74.483, E3 +36321.208}
SPL {X  -136.371, Y  +755.165, Z    +0.000, E1   -74.152, E3 +36326.753}
SPL {X  -133.102, Y  +760.274, Z    +0.000, E1   -73.777, E3 +36332.139}
SPL {X  -128.975, Y  +766.169, Z    +0.000, E1   -73.313, E3 +36338.414}
SPL {X  -124.947, Y  +771.425, Z    +0.000, E1   -72.782, E3 +36344.107}
SPL {X  -121.698, Y  +775.357, Z    +0.000, E1   -72.353, E3 +36348.301}
SPL {X  -118.622, Y  +778.858, Z    +0.000, E1   -71.924, E3 +36351.927}
SPL {X   -66.171, Y  +817.165, Z    +0.000, E1   -56.016, E3 +36503.286}
ENDSPLINE

SPLINE
SPL {X  -126.418, Y  +769.557, Z    +0.000, E1   -57.118, E3 +36686.527}
SPL {X  -148.476, Y  +731.097, Z    +0.000, E1   -47.824, E3 +36701.683}
SPL {X  -156.642, Y  +704.059, Z    +0.000, E1   -33.659, E3 +36706.325}
SPL {X  -159.317, Y  +686.157, Z    +0.000, E1   -18.660, E3 +36707.815}
SPL {X  -159.973, Y  +673.799, Z    +0.000, E1    -5.345, E3 +36708.264}
SPL {X  -159.990, Y  +669.500, Z    +0.000, E1    +0.000, E3 +36708.304}
SPL {X  -159.990, Y  +667.794, Z    +0.000, E1    +4.255, E3 +36708.315}
SPL {X  -159.990, Y  +664.091, Z    +0.000, E1   +14.928, E3 +36708.387}
SPL {X  -159.990, Y  +659.599, Z    +0.000, E1   +28.016, E3 +36708.557}
SPL {X  -159.990, Y  +652.711, Z    +0.000, E1   +44.293, E3 +36709.037}
SPL {X  -159.990, Y  +640.730, Z    +0.000, E1   +60.297, E3 +36710.386}
SPL {X  -159.990, Y  +620.478, Z    +0.000, E1   +70.026, E3 +36714.199}
SPL {X  -159.990, Y  +573.021, Z    +0.000, E1   +74.619, E3 +36728.143}
SPL {X  -154.165, Y  +339.724, Z    +0.000, E1   +75.927, E3 +36823.990}
SPL {X  -150.223, Y  +327.456, Z    +0.000, E1   +75.573, E3 +36834.255}
SPL {X  -136.549, Y  +299.126, Z    +0.000, E1   +77.537, E3 +36827.145}
ENDSPLINE

SPLINE
SPL {X  -136.862, Y  +299.641, Z    +0.000, E1   +76.604, E3 +36835.787}
ENDSPLINE

SPLINE
SPL {X  -136.434, Y  +298.938, Z    +0.000, E1   +75.982, E3 +36841.678}
SPL {X  -135.890, Y  +298.057, Z    +0.000, E1   +75.040, E3 +36850.144}
SPL {X  -134.349, Y  +295.626, Z    +0.000, E1   +74.322, E3 +36856.991}
SPL {X  -131.287, Y  +291.064, Z    +0.000, E1   +73.972, E3 +36861.804}
SPL {X  -128.265, Y  +286.871, Z    +0.000, E1   +73.613, E3 +36866.260}
SPL {X  -125.161, Y  +282.843, Z    +0.000, E1   +73.232, E3 +36870.531}
SPL {X  -122.038, Y  +279.042, Z    +0.000, E1   +72.832, E3 +36874.511}
SPL {X  -118.642, Y  +275.165, Z    +0.000, E1   +72.381, E3 +36878.474}
SPL {X   -66.040, Y  +236.776, Z    +0.000, E1   +55.694, E3 +37039.838}
ENDSPLINE

SPLINE
SPL {X  -127.452, Y  +285.790, Z    +0.000, E1   +56.591, E3 +37213.783}
SPL {X  -151.591, Y  +331.344, Z    +0.000, E1   +43.870, E3 +37229.883}
SPL {X  -158.135, Y  +358.205, Z    +0.000, E1   +26.984, E3 +37233.610}
SPL {X  -159.602, Y  +371.361, Z    +0.000, E1   +14.835, E3 +37234.506}
SPL {X  -159.981, Y  +380.818, Z    +0.000, E1    +4.512, E3 +37234.784}
SPL {X  -159.990, Y  +384.681, Z    +0.000, E1    -0.222, E3 +37234.813}
SPL {X  -159.990, Y  +387.626, Z    +0.000, E1    -8.190, E3 +37234.841}
SPL {X  -159.990, Y  +390.340, Z    +0.000, E1   -15.987, E3 +37234.906}
SPL {X  -159.990, Y  +394.216, Z    +0.000, E1   -27.062, E3 +37235.068}
SPL {X  -159.990, Y  +399.855, Z    +0.000, E1   -40.916, E3 +37235.439}
SPL {X  -159.990, Y  +405.475, Z    +0.000, E1   -51.039, E3 +37235.956}
SPL {X  -159.990, Y  +414.231, Z    +0.000, E1   -60.575, E3 +37237.140}
SPL {X  -159.990, Y  +462.953, Z    +0.000, E1   -73.611, E3 +37248.879}
SPL {X  -153.839, Y  +715.436, Z    +0.000, E1   -75.884, E3 +37351.310}
SPL {X  -149.923, Y  +727.355, Z    +0.000, E1   -75.515, E3 +37361.419}
SPL {X  -145.995, Y  +736.939, Z    +0.000, E1   -75.150, E3 +37370.154}
SPL {X  -141.012, Y  +747.080, Z    +0.000, E1   -74.661, E3 +37380.006}
SPL {X  -136.371, Y  +755.165, Z    +0.000, E1   -74.152, E3 +37388.292}
SPL {X  -133.102, Y  +760.274, Z    +0.000, E1   -73.777, E3 +37393.677}
SPL {X  -128.975, Y  +766.169, Z    +0.000, E1   -73.313, E3 +37399.952}
SPL {X  -124.947, Y  +771.425, Z    +0.000, E1   -72.782, E3 +37405.645}
SPL {X  -121.698, Y  +775.357, Z    +0.000, E1   -72.353, E3 +37409.840}
SPL {X  -118.622, Y  +778.858, Z    +0.000, E1   -71.924, E3 +37413.466}
SPL {X   -66.171, Y  +817.165, Z    +0.000, E1   -56.016, E3 +37564.824}
ENDSPLINE

SPLINE
SPL {X  -126.418, Y  +769.557, Z    +0.000, E1   -57.118, E3 +37748.065}
SPL {X  -148.476, Y  +731.097, Z    +0.000, E1   -47.824, E3 +37763.221}
SPL {X  -156.642, Y  +704.059, Z    +0.000, E1   -33.659, E3 +37767.863}
SPL {X  -159.317, Y  +686.157, Z    +0.000, E1   -18.660, E3 +37769.353}
SPL {X  -159.907, Y  +676.666, Z    +0.000, E1    -8.555, E3 +37769.751}
SPL {X  -159.990, Y  +669.586, Z    +0.000, E1    -0.216, E3 +37769.842}
SPL {X  -159.990, Y  +667.794, Z    +0.000, E1    +4.255, E3 +37769.853}
SPL {X  -159.990, Y  +664.091, Z    +0.000, E1   +14.928, E3 +37769.925}
SPL {X  -159.990, Y  +659.599, Z    +0.000, E1   +28.016, E3 +37770.096}
SPL {X  -159.990, Y  +652.711, Z    +0.000, E1   +44.293, E3 +37770.575}
SPL {X  -159.990, Y  +640.730, Z    +0.000, E1   +60.297, E3 +37771.924}
SPL {X  -159.990, Y  +620.478, Z    +0.000, E1   +70.026, E3 +37775.738}
SPL {X  -159.990, Y  +573.021, Z    +0.000, E1   +74.619, E3 +37789.681}
SPL {X  -154.165, Y  +339.724, Z    +0.000, E1   +75.927, E3 +37885.528}
SPL {X  -150.223, Y  +327.456, Z    +0.000, E1   +75.573, E3 +37895.793}
SPL {X  -136.549, Y  +299.126, Z    +0.000, E1   +77.537, E3 +37888.683}
ENDSPLINE

SPLINE
SPL {X  -136.862, Y  +299.641, Z    +0.000, E1   +76.604, E3 +37897.325}
ENDSPLINE

SPLINE
SPL {X  -136.434, Y  +298.938, Z    +0.000, E1   +75.982, E3 +37903.216}
SPL {X  -135.890, Y  +298.057, Z    +0.000, E1   +75.040, E3 +37911.682}
SPL {X  -134.349, Y  +295.626, Z    +0.000, E1   +74.322, E3 +37918.530}
SPL {X  -131.287, Y  +291.064, Z    +0.000, E1   +73.972, E3 +37923.342}
SPL {X  -128.265, Y  +286.871, Z    +0.000, E1   +73.613, E3 +37927.798}
SPL {X  -125.161, Y  +282.843, Z    +0.000, E1   +73.232, E3 +37932.070}
SPL {X  -122.038, Y  +279.042, Z    +0.000, E1   +72.832, E3 +37936.050}
SPL {X  -118.642, Y  +275.165, Z    +0.000, E1   +72.381, E3 +37940.013}
SPL {X   -66.040, Y  +236.776, Z    +0.000, E1   +55.694, E3 +38101.376}
ENDSPLINE

SPLINE
SPL {X  -127.452, Y  +285.790, Z    +0.000, E1   +56.591, E3 +38275.322}
SPL {X  -148.001, Y  +321.733, Z    +0.000, E1   +47.810, E3 +38289.425}
SPL {X  -154.604, Y  +341.337, Z    +0.000, E1   +38.630, E3 +38293.199}
SPL {X  -158.135, Y  +358.205, Z    +0.000, E1   +26.984, E3 +38295.149}
SPL {X  -159.602, Y  +371.361, Z    +0.000, E1   +14.835, E3 +38296.045}
SPL {X  -159.981, Y  +380.818, Z    +0.000, E1    +4.512, E3 +38296.322}
SPL {X  -159.990, Y  +384.681, Z    +0.000, E1    -0.222, E3 +38296.351}
SPL {X  -159.990, Y  +389.079, Z    +0.000, E1   -12.017, E3 +38296.414}
SPL {X  -159.990, Y  +394.216, Z    +0.000, E1   -27.062, E3 +38296.606}
SPL {X  -159.990, Y  +399.855, Z    +0.000, E1   -40.916, E3 +38296.977}
SPL {X  -159.990, Y  +405.475, Z    +0.000, E1   -51.039, E3 +38297.494}
SPL {X  -159.990, Y  +414.231, Z    +0.000, E1   -60.575, E3 +38298.678}
SPL {X  -159.990, Y  +462.953, Z    +0.000, E1   -73.611, E3 +38310.417}
SPL {X  -153.839, Y  +715.436, Z    +0.000, E1   -75.884, E3 +38412.848}
SPL {X  -148.840, Y  +730.182, Z    +0.000, E1   -75.434, E3 +38425.425}
SPL {X  -143.409, Y  +742.426, Z    +0.000, E1   -74.905, E3 +38436.937}
SPL {X  -139.557, Y  +749.735, Z    +0.000, E1   -74.483, E3 +38444.285}
SPL {X  -136.371, Y  +755.165, Z    +0.000, E1   -74.152, E3 +38449.830}
SPL {X  -133.102, Y  +760.274, Z    +0.000, E1   -73.777, E3 +38455.215}
SPL {X  -128.975, Y  +766.169, Z    +0.000, E1   -73.313, E3 +38461.491}
SPL {X  -124.947, Y  +771.425, Z    +0.000, E1   -72.782, E3 +38467.184}
SPL {X  -121.698, Y  +775.357, Z    +0.000, E1   -72.353, E3 +38471.378}
SPL {X  -118.622, Y  +778.858, Z    +0.000, E1   -71.924, E3 +38475.004}
SPL {X   -66.171, Y  +817.165, Z    +0.000, E1   -56.016, E3 +38626.363}
ENDSPLINE

SPLINE
SPL {X  -126.418, Y  +769.557, Z    +0.000, E1   -57.118, E3 +38809.604}
SPL {X  -145.244, Y  +738.589, Z    +0.000, E1   -50.405, E3 +38822.845}
SPL {X  -150.151, Y  +726.741, Z    +0.000, E1   -46.068, E3 +38825.772}
SPL {X  -156.642, Y  +704.059, Z    +0.000, E1   -33.659, E3 +38829.402}
SPL {X  -159.317, Y  +686.157, Z    +0.000, E1   -18.660, E3 +38830.892}
SPL {X  -159.973, Y  +673.799, Z    +0.000, E1    -5.345, E3 +38831.340}
SPL {X  -159.990, Y  +669.500, Z    +0.000, E1    +0.000, E3 +38831.381}
SPL {X  -159.990, Y  +667.794, Z    +0.000, E1    +4.255, E3 +38831.392}
SPL {X  -159.990, Y  +664.091, Z    +0.000, E1   +14.928, E3 +38831.464}
SPL {X  -159.990, Y  +658.301, Z    +0.000, E1   +31.283, E3 +38831.716}
SPL {X  -159.990, Y  +650.845, Z    +0.000, E1   +47.892, E3 +38832.262}
SPL {X  -159.990, Y  +640.730, Z    +0.000, E1   +60.297, E3 +38833.463}
SPL {X  -159.990, Y  +620.478, Z    +0.000, E1   +70.026, E3 +38837.276}
SPL {X  -159.990, Y  +573.021, Z    +0.000, E1   +74.619, E3 +38851.220}
SPL {X  -154.165, Y  +339.724, Z    +0.000, E1   +75.927, E3 +38947.067}
SPL {X  -150.223, Y  +327.456, Z    +0.000, E1   +75.573, E3 +38957.332}
SPL {X  -136.549, Y  +299.126, Z    +0.000, E1   +77.537, E3 +38950.222}
ENDSPLINE

SPLINE
SPL {X  -136.862, Y  +299.641, Z    +0.000, E1   +76.604, E3 +38958.864}
ENDSPLINE

SPLINE
SPL {X  -136.434, Y  +298.938, Z    +0.000, E1   +75.982, E3 +38964.755}
SPL {X  -135.890, Y  +298.057, Z    +0.000, E1   +75.040, E3 +38973.221}
SPL {X  -134.349, Y  +295.626, Z    +0.000, E1   +74.322, E3 +38980.068}
SPL {X  -131.287, Y  +291.064, Z    +0.000, E1   +73.972, E3 +38984.881}
SPL {X  -128.265, Y  +286.871, Z    +0.000, E1   +73.613, E3 +38989.337}
SPL {X  -125.161, Y  +282.843, Z    +0.000, E1   +73.232, E3 +38993.608}
SPL {X  -122.038, Y  +279.042, Z    +0.000, E1   +72.832, E3 +38997.588}
SPL {X  -118.642, Y  +275.165, Z    +0.000, E1   +72.381, E3 +39001.551}
SPL {X   -66.040, Y  +236.776, Z    +0.000, E1   +55.694, E3 +39162.915}
ENDSPLINE

SPLINE
SPL {X  -127.452, Y  +285.790, Z    +0.000, E1   +56.591, E3 +39336.860}
SPL {X  -148.001, Y  +321.733, Z    +0.000, E1   +47.810, E3 +39350.964}
SPL {X  -154.604, Y  +341.337, Z    +0.000, E1   +38.630, E3 +39354.737}
SPL {X  -158.135, Y  +358.205, Z    +0.000, E1   +26.984, E3 +39356.687}
SPL {X  -159.602, Y  +371.361, Z    +0.000, E1   +14.835, E3 +39357.583}
SPL {X  -159.981, Y  +380.818, Z    +0.000, E1    +4.512, E3 +39357.861}
SPL {X  -159.990, Y  +384.681, Z    +0.000, E1    -0.222, E3 +39357.890}
SPL {X  -159.990, Y  +389.079, Z    +0.000, E1   -12.017, E3 +39357.953}
SPL {X  -159.990, Y  +394.216, Z    +0.000, E1   -27.062, E3 +39358.145}
SPL {X  -159.990, Y  +399.855, Z    +0.000, E1   -40.916, E3 +39358.516}
SPL {X  -159.990, Y  +405.475, Z    +0.000, E1   -51.039, E3 +39359.033}
SPL {X  -159.990, Y  +414.231, Z    +0.000, E1   -60.575, E3 +39360.217}
SPL {X  -159.990, Y  +462.953, Z    +0.000, E1   -73.611, E3 +39371.956}
SPL {X  -153.839, Y  +715.436, Z    +0.000, E1   -75.884, E3 +39474.386}
SPL {X  -148.840, Y  +730.182, Z    +0.000, E1   -75.434, E3 +39486.963}
SPL {X  -143.409, Y  +742.426, Z    +0.000, E1   -74.905, E3 +39498.475}
SPL {X  -139.557, Y  +749.735, Z    +0.000, E1   -74.483, E3 +39505.823}
SPL {X  -136.371, Y  +755.165, Z    +0.000, E1   -74.152, E3 +39511.369}
SPL {X  -133.102, Y  +760.274, Z    +0.000, E1   -73.777, E3 +39516.754}
SPL {X  -128.975, Y  +766.169, Z    +0.000, E1   -73.313, E3 +39523.029}
SPL {X  -124.947, Y  +771.425, Z    +0.000, E1   -72.782, E3 +39528.722}
SPL {X  -121.698, Y  +775.357, Z    +0.000, E1   -72.353, E3 +39532.917}
SPL {X  -118.622, Y  +778.858, Z    +0.000, E1   -71.924, E3 +39536.543}
SPL {X   -66.171, Y  +817.165, Z    +0.000, E1   -56.016, E3 +39687.901}
ENDSPLINE

SPLINE
SPL {X  -126.418, Y  +769.557, Z    +0.000, E1   -57.118, E3 +39871.142}
SPL {X  -145.244, Y  +738.589, Z    +0.000, E1   -50.405, E3 +39884.384}
SPL {X  -150.151, Y  +726.741, Z    +0.000, E1   -46.068, E3 +39887.311}
SPL {X  -156.642, Y  +704.059, Z    +0.000, E1   -33.659, E3 +39890.940}
SPL {X  -159.317, Y  +686.157, Z    +0.000, E1   -18.660, E3 +39892.430}
SPL {X  -159.973, Y  +673.799, Z    +0.000, E1    -5.345, E3 +39892.879}
SPL {X  -159.990, Y  +669.500, Z    +0.000, E1    +0.000, E3 +39892.919}
SPL {X  -159.990, Y  +667.794, Z    +0.000, E1    +4.255, E3 +39892.930}
SPL {X  -159.990, Y  +664.091, Z    +0.000, E1   +14.928, E3 +39893.002}
SPL {X  -159.990, Y  +658.301, Z    +0.000, E1   +31.283, E3 +39893.255}
SPL {X  -159.990, Y  +650.845, Z    +0.000, E1   +47.892, E3 +39893.800}
SPL {X  -159.990, Y  +640.730, Z    +0.000, E1   +60.297, E3 +39895.001}
SPL {X  -159.990, Y  +620.478, Z    +0.000, E1   +70.026, E3 +39898.814}
SPL {X  -159.990, Y  +573.021, Z    +0.000, E1   +74.619, E3 +39912.758}
SPL {X  -154.165, Y  +339.724, Z    +0.000, E1   +75.927, E3 +40008.605}
SPL {X  -150.223, Y  +327.456, Z    +0.000, E1   +75.573, E3 +40018.870}
SPL {X  -136.549, Y  +299.126, Z    +0.000, E1   +77.537, E3 +40011.760}
ENDSPLINE

SPLINE
SPL {X  -136.862, Y  +299.641, Z    +0.000, E1   +76.604, E3 +40020.402}
ENDSPLINE

SPLINE
SPL {X  -136.434, Y  +298.938, Z    +0.000, E1   +75.982, E3 +40026.293}
SPL {X  -135.890, Y  +298.057, Z    +0.000, E1   +75.040, E3 +40034.759}
SPL {X  -134.349, Y  +295.626, Z    +0.000, E1   +74.322, E3 +40041.606}
SPL {X  -131.287, Y  +291.064, Z    +0.000, E1   +73.972, E3 +40046.419}
SPL {X  -128.265, Y  +286.871, Z    +0.000, E1   +73.613, E3 +40050.875}
SPL {X  -125.161, Y  +282.843, Z    +0.000, E1   +73.232, E3 +40055.147}
SPL {X  -122.038, Y  +279.042, Z    +0.000, E1   +72.832, E3 +40059.127}
SPL {X  -118.642, Y  +275.165, Z    +0.000, E1   +72.381, E3 +40063.090}
SPL {X   -66.040, Y  +236.776, Z    +0.000, E1   +55.694, E3 +40224.453}
ENDSPLINE

SPLINE
SPL {X  -127.452, Y  +285.790, Z    +0.000, E1   +56.591, E3 +40398.399}
SPL {X  -148.001, Y  +321.733, Z    +0.000, E1   +47.810, E3 +40412.502}
SPL {X  -154.604, Y  +341.337, Z    +0.000, E1   +38.630, E3 +40416.276}
SPL {X  -158.135, Y  +358.205, Z    +0.000, E1   +26.984, E3 +40418.226}
SPL {X  -159.602, Y  +371.361, Z    +0.000, E1   +14.835, E3 +40419.122}
SPL {X  -159.981, Y  +380.818, Z    +0.000, E1    +4.512, E3 +40419.399}
SPL {X  -159.990, Y  +384.681, Z    +0.000, E1    -0.222, E3 +40419.428}
SPL {X  -159.990, Y  +389.079, Z    +0.000, E1   -12.017, E3 +40419.491}
SPL {X  -159.990, Y  +394.216, Z    +0.000, E1   -27.062, E3 +40419.683}
SPL {X  -159.990, Y  +399.855, Z    +0.000, E1   -40.916, E3 +40420.054}
SPL {X  -159.990, Y  +405.475, Z    +0.000, E1   -51.039, E3 +40420.571}
SPL {X  -159.990, Y  +414.231, Z    +0.000, E1   -60.575, E3 +40421.755}
SPL {X  -159.990, Y  +462.953, Z    +0.000, E1   -73.611, E3 +40433.494}
SPL {X  -153.839, Y  +715.436, Z    +0.000, E1   -75.884, E3 +40535.925}
SPL {X  -148.840, Y  +730.182, Z    +0.000, E1   -75.434, E3 +40548.502}
SPL {X  -143.409, Y  +742.426, Z    +0.000, E1   -74.905, E3 +40560.014}
SPL {X  -139.557, Y  +749.735, Z    +0.000, E1   -74.483, E3 +40567.362}
SPL {X  -136.371, Y  +755.165, Z    +0.000, E1   -74.152, E3 +40572.907}
SPL {X  -133.102, Y  +760.274, Z    +0.000, E1   -73.777, E3 +40578.292}
SPL {X  -128.975, Y  +766.169, Z    +0.000, E1   -73.313, E3 +40584.568}
SPL {X  -124.947, Y  +771.425, Z    +0.000, E1   -72.782, E3 +40590.261}
SPL {X  -121.698, Y  +775.357, Z    +0.000, E1   -72.353, E3 +40594.455}
SPL {X  -118.622, Y  +778.858, Z    +0.000, E1   -71.924, E3 +40598.081}
SPL {X   -66.171, Y  +817.165, Z    +0.000, E1   -56.016, E3 +40749.440}
ENDSPLINE

SPLINE
SPL {X  -126.418, Y  +769.557, Z    +0.000, E1   -57.118, E3 +40932.681}
SPL {X  -145.244, Y  +738.589, Z    +0.000, E1   -50.405, E3 +40945.922}
SPL {X  -150.151, Y  +726.741, Z    +0.000, E1   -46.068, E3 +40948.849}
SPL {X  -156.642, Y  +704.059, Z    +0.000, E1   -33.659, E3 +40952.479}
SPL {X  -159.317, Y  +686.157, Z    +0.000, E1   -18.660, E3 +40953.969}
SPL {X  -159.973, Y  +673.799, Z    +0.000, E1    -5.345, E3 +40954.417}
SPL {X  -159.990, Y  +669.500, Z    +0.000, E1    +0.000, E3 +40954.457}
SPL {X  -159.990, Y  +667.794, Z    +0.000, E1    +4.255, E3 +40954.469}
SPL {X  -159.990, Y  +664.091, Z    +0.000, E1   +14.928, E3 +40954.541}
SPL {X  -159.990, Y  +658.301, Z    +0.000, E1   +31.283, E3 +40954.793}
SPL {X  -159.990, Y  +650.845, Z    +0.000, E1   +47.892, E3 +40955.338}
SPL {X  -159.990, Y  +640.730, Z    +0.000, E1   +60.297, E3 +40956.540}
SPL {X  -159.990, Y  +620.478, Z    +0.000, E1   +70.026, E3 +40960.353}
SPL {X  -159.990, Y  +573.021, Z    +0.000, E1   +74.619, E3 +40974.297}
SPL {X  -154.165, Y  +339.724, Z    +0.000, E1   +75.927, E3 +41070.144}
SPL {X  -150.223, Y  +327.456, Z    +0.000, E1   +75.573, E3 +41080.409}
SPL {X  -136.549, Y  +299.126, Z    +0.000, E1   +77.537, E3 +41073.299}
ENDSPLINE

SPLINE
SPL {X  -136.626, Y  +299.252, Z    +0.000, E1   +76.314, E3 +41084.949}
ENDSPLINE

SPLINE
SPL {X  -135.890, Y  +298.057, Z    +0.000, E1   +75.040, E3 +41096.298}
SPL {X  -134.349, Y  +295.626, Z    +0.000, E1   +74.322, E3 +41103.145}
SPL {X  -131.287, Y  +291.064, Z    +0.000, E1   +73.972, E3 +41107.957}
SPL {X  -128.265, Y  +286.871, Z    +0.000, E1   +73.613, E3 +41112.413}
SPL {X  -125.161, Y  +282.843, Z    +0.000, E1   +73.232, E3 +41116.685}
SPL {X  -122.038, Y  +279.042, Z    +0.000, E1   +72.832, E3 +41120.665}
SPL {X  -118.642, Y  +275.165, Z    +0.000, E1   +72.381, E3 +41124.628}
SPL {X   -66.040, Y  +236.776, Z    +0.000, E1   +55.694, E3 +41285.992}
ENDSPLINE

SPLINE
SPL {X  -127.452, Y  +285.790, Z    +0.000, E1   +56.591, E3 +41459.937}
SPL {X  -151.591, Y  +331.344, Z    +0.000, E1   +43.870, E3 +41476.036}
SPL {X  -158.135, Y  +358.205, Z    +0.000, E1   +26.984, E3 +41479.764}
SPL {X  -159.602, Y  +371.361, Z    +0.000, E1   +14.835, E3 +41480.660}
SPL {X  -159.981, Y  +380.818, Z    +0.000, E1    +4.512, E3 +41480.938}
SPL {X  -159.990, Y  +384.681, Z    +0.000, E1    -0.222, E3 +41480.967}
SPL {X  -159.990, Y  +387.626, Z    +0.000, E1    -8.190, E3 +41480.995}
SPL {X  -159.990, Y  +390.340, Z    +0.000, E1   -15.987, E3 +41481.060}
SPL {X  -159.990, Y  +394.216, Z    +0.000, E1   -27.062, E3 +41481.222}
SPL {X  -159.990, Y  +399.855, Z    +0.000, E1   -40.916, E3 +41481.593}
SPL {X  -159.990, Y  +405.475, Z    +0.000, E1   -51.039, E3 +41482.110}
SPL {X  -159.990, Y  +414.231, Z    +0.000, E1   -60.575, E3 +41483.294}
SPL {X  -159.990, Y  +462.953, Z    +0.000, E1   -73.611, E3 +41495.033}
SPL {X  -153.839, Y  +715.436, Z    +0.000, E1   -75.884, E3 +41597.463}
SPL {X  -149.923, Y  +727.355, Z    +0.000, E1   -75.515, E3 +41607.573}
SPL {X  -145.995, Y  +736.939, Z    +0.000, E1   -75.150, E3 +41616.308}
SPL {X  -142.305, Y  +744.618, Z    +0.000, E1   -74.773, E3 +41623.752}
SPL {X  -139.557, Y  +749.735, Z    +0.000, E1   -74.483, E3 +41628.900}
SPL {X  -136.371, Y  +755.165, Z    +0.000, E1   -74.152, E3 +41634.446}
SPL {X  -131.455, Y  +762.694, Z    +0.000, E1   -73.615, E3 +41642.364}
SPL {X  -125.933, Y  +770.180, Z    +0.000, E1   -72.934, E3 +41650.428}
SPL {X  -121.698, Y  +775.357, Z    +0.000, E1   -72.353, E3 +41655.994}
SPL {X  -118.622, Y  +778.858, Z    +0.000, E1   -71.924, E3 +41659.620}
SPL {X   -66.171, Y  +817.165, Z    +0.000, E1   -56.016, E3 +41810.978}
ENDSPLINE

SPLINE
SPL {X  -126.418, Y  +769.557, Z    +0.000, E1   -57.118, E3 +41994.219}
SPL {X  -145.244, Y  +738.589, Z    +0.000, E1   -50.405, E3 +42007.461}
SPL {X  -150.151, Y  +726.741, Z    +0.000, E1   -46.068, E3 +42010.388}
SPL {X  -156.642, Y  +704.059, Z    +0.000, E1   -33.659, E3 +42014.017}
SPL {X  -159.317, Y  +686.157, Z    +0.000, E1   -18.660, E3 +42015.507}
SPL {X  -159.973, Y  +673.799, Z    +0.000, E1    -5.345, E3 +42015.956}
SPL {X  -159.990, Y  +669.500, Z    +0.000, E1    +0.000, E3 +42015.996}
SPL {X  -159.990, Y  +667.794, Z    +0.000, E1    +4.255, E3 +42016.007}
SPL {X  -159.990, Y  +664.091, Z    +0.000, E1   +14.928, E3 +42016.079}
SPL {X  -159.990, Y  +659.599, Z    +0.000, E1   +28.016, E3 +42016.250}
SPL {X  -159.990, Y  +652.711, Z    +0.000, E1   +44.293, E3 +42016.729}
SPL {X  -159.990, Y  +640.730, Z    +0.000, E1   +60.297, E3 +42018.078}
SPL {X  -159.990, Y  +620.478, Z    +0.000, E1   +70.026, E3 +42021.891}
SPL {X  -159.990, Y  +573.021, Z    +0.000, E1   +74.619, E3 +42035.835}
SPL {X  -154.165, Y  +339.724, Z    +0.000, E1   +75.927, E3 +42131.682}
SPL {X  -150.571, Y  +328.416, Z    +0.000, E1   +75.599, E3 +42141.127}
SPL {X  -148.206, Y  +322.236, Z    +0.000, E1   +75.365, E3 +42146.672}
SPL {X  -136.549, Y  +299.126, Z    +0.000, E1   +77.537, E3 +42134.837}
ENDSPLINE

SPLINE
SPL {X  -136.862, Y  +299.641, Z    +0.000, E1   +76.604, E3 +42143.479}
ENDSPLINE

SPLINE
SPL {X  -136.434, Y  +298.938, Z    +0.000, E1   +75.982, E3 +42149.370}
SPL {X  -135.890, Y  +298.057, Z    +0.000, E1   +75.040, E3 +42157.836}
SPL {X  -134.349, Y  +295.626, Z    +0.000, E1   +74.322, E3 +42164.683}
SPL {X  -131.287, Y  +291.064, Z    +0.000, E1   +73.972, E3 +42169.496}
SPL {X  -128.265, Y  +286.871, Z    +0.000, E1   +73.613, E3 +42173.952}
SPL {X  -125.161, Y  +282.843, Z    +0.000, E1   +73.232, E3 +42178.224}
SPL {X  -122.038, Y  +279.042, Z    +0.000, E1   +72.832, E3 +42182.204}
SPL {X  -118.642, Y  +275.165, Z    +0.000, E1   +72.381, E3 +42186.167}
SPL {X   -66.040, Y  +236.776, Z    +0.000, E1   +55.694, E3 +42347.530}
ENDSPLINE

SPLINE
SPL {X  -127.452, Y  +285.790, Z    +0.000, E1   +56.591, E3 +42521.476}
SPL {X  -151.591, Y  +331.344, Z    +0.000, E1   +43.870, E3 +42537.575}
SPL {X  -158.135, Y  +358.205, Z    +0.000, E1   +26.984, E3 +42541.302}
SPL {X  -159.602, Y  +371.361, Z    +0.000, E1   +14.835, E3 +42542.198}
SPL {X  -159.981, Y  +380.818, Z    +0.000, E1    +4.512, E3 +42542.476}
SPL {X  -159.990, Y  +384.681, Z    +0.000, E1    -0.222, E3 +42542.505}
SPL {X  -159.990, Y  +389.079, Z    +0.000, E1   -12.017, E3 +42542.568}
SPL {X  -159.990, Y  +394.216, Z    +0.000, E1   -27.062, E3 +42542.760}
SPL {X  -159.990, Y  +399.855, Z    +0.000, E1   -40.916, E3 +42543.131}
SPL {X  -159.990, Y  +405.475, Z    +0.000, E1   -51.039, E3 +42543.648}
SPL {X  -159.990, Y  +414.231, Z    +0.000, E1   -60.575, E3 +42544.832}
SPL {X  -159.990, Y  +462.953, Z    +0.000, E1   -73.611, E3 +42556.571}
SPL {X  -153.839, Y  +715.436, Z    +0.000, E1   -75.884, E3 +42659.002}
SPL {X  -148.840, Y  +730.182, Z    +0.000, E1   -75.434, E3 +42671.578}
SPL {X  -143.409, Y  +742.426, Z    +0.000, E1   -74.905, E3 +42683.090}
SPL {X  -139.557, Y  +749.735, Z    +0.000, E1   -74.483, E3 +42690.439}
SPL {X  -136.371, Y  +755.165, Z    +0.000, E1   -74.152, E3 +42695.984}
SPL {X  -133.102, Y  +760.274, Z    +0.000, E1   -73.777, E3 +42701.369}
SPL {X  -128.975, Y  +766.169, Z    +0.000, E1   -73.313, E3 +42707.645}
SPL {X  -124.947, Y  +771.425, Z    +0.000, E1   -72.782, E3 +42713.338}
SPL {X  -121.698, Y  +775.357, Z    +0.000, E1   -72.353, E3 +42717.532}
SPL {X  -118.622, Y  +778.858, Z    +0.000, E1   -71.924, E3 +42721.158}
SPL {X   -66.171, Y  +817.165, Z    +0.000, E1   -56.016, E3 +42872.517}
ENDSPLINE

SPLINE
SPL {X  -126.418, Y  +769.557, Z    +0.000, E1   -57.118, E3 +43055.758}
SPL {X  -145.244, Y  +738.589, Z    +0.000, E1   -50.405, E3 +43068.999}
SPL {X  -150.151, Y  +726.741, Z    +0.000, E1   -46.068, E3 +43071.926}
SPL {X  -156.642, Y  +704.059, Z    +0.000, E1   -33.659, E3 +43075.555}
SPL {X  -159.317, Y  +686.157, Z    +0.000, E1   -18.660, E3 +43077.046}
SPL {X  -159.973, Y  +673.799, Z    +0.000, E1    -5.345, E3 +43077.494}
SPL {X  -159.990, Y  +669.500, Z    +0.000, E1    +0.000, E3 +43077.534}
SPL {X  -159.990, Y  +667.794, Z    +0.000, E1    +4.255, E3 +43077.546}
SPL {X  -159.990, Y  +664.091, Z    +0.000, E1   +14.928, E3 +43077.618}
SPL {X  -159.990, Y  +658.301, Z    +0.000, E1   +31.283, E3 +43077.870}
SPL {X  -159.990, Y  +650.845, Z    +0.000, E1   +47.892, E3 +43078.415}
SPL {X  -159.990, Y  +640.730, Z    +0.000, E1   +60.297, E3 +43079.617}
SPL {X  -159.990, Y  +620.478, Z    +0.000, E1   +70.026, E3 +43083.430}
SPL {X  -159.990, Y  +573.021, Z    +0.000, E1   +74.619, E3 +43097.374}
SPL {X  -154.165, Y  +339.724, Z    +0.000, E1   +75.927, E3 +43193.221}
SPL {X  -150.223, Y  +327.456, Z    +0.000, E1   +75.573, E3 +43203.486}
SPL {X  -136.549, Y  +299.126, Z    +0.000, E1   +77.537, E3 +43196.376}
ENDSPLINE

SPLINE
SPL {X  -136.862, Y  +299.641, Z    +0.000, E1   +76.604, E3 +43205.018}
ENDSPLINE

SPLINE
SPL {X  -136.434, Y  +298.938, Z    +0.000, E1   +75.982, E3 +43210.909}
SPL {X  -135.890, Y  +298.057, Z    +0.000, E1   +75.040, E3 +43219.375}
SPL {X  -134.349, Y  +295.626, Z    +0.000, E1   +74.322, E3 +43226.222}
SPL {X  -131.287, Y  +291.064, Z    +0.000, E1   +73.972, E3 +43231.034}
SPL {X  -128.265, Y  +286.871, Z    +0.000, E1   +73.613, E3 +43235.490}
SPL {X  -125.161, Y  +282.843, Z    +0.000, E1   +73.232, E3 +43239.762}
SPL {X  -122.038, Y  +279.042, Z    +0.000, E1   +72.832, E3 +43243.742}
SPL {X  -118.642, Y  +275.165, Z    +0.000, E1   +72.381, E3 +43247.705}
SPL {X   -66.040, Y  +236.776, Z    +0.000, E1   +55.694, E3 +43409.069}
ENDSPLINE

SPLINE
SPL {X  -127.452, Y  +285.790, Z    +0.000, E1   +56.591, E3 +43583.014}
SPL {X  -151.591, Y  +331.344, Z    +0.000, E1   +43.870, E3 +43599.113}
SPL {X  -158.135, Y  +358.205, Z    +0.000, E1   +26.984, E3 +43602.841}
SPL {X  -159.602, Y  +371.361, Z    +0.000, E1   +14.835, E3 +43603.737}
SPL {X  -159.981, Y  +380.818, Z    +0.000, E1    +4.512, E3 +43604.015}
SPL {X  -159.990, Y  +384.681, Z    +0.000, E1    -0.222, E3 +43604.044}
SPL {X  -159.990, Y  +387.626, Z    +0.000, E1    -8.190, E3 +43604.072}
SPL {X  -159.990, Y  +390.340, Z    +0.000, E1   -15.987, E3 +43604.137}
SPL {X  -159.990, Y  +394.216, Z    +0.000, E1   -27.062, E3 +43604.299}
SPL {X  -159.990, Y  +399.855, Z    +0.000, E1   -40.916, E3 +43604.670}
SPL {X  -159.990, Y  +405.475, Z    +0.000, E1   -51.039, E3 +43605.187}
SPL {X  -159.990, Y  +414.231, Z    +0.000, E1   -60.575, E3 +43606.371}
SPL {X  -159.990, Y  +462.953, Z    +0.000, E1   -73.611, E3 +43618.110}
SPL {X  -153.839, Y  +715.436, Z    +0.000, E1   -75.884, E3 +43720.540}
SPL {X  -148.840, Y  +730.182, Z    +0.000, E1   -75.434, E3 +43733.117}
SPL {X  -143.409, Y  +742.426, Z    +0.000, E1   -74.905, E3 +43744.629}
SPL {X  -139.557, Y  +749.735, Z    +0.000, E1   -74.483, E3 +43751.977}
SPL {X  -136.371, Y  +755.165, Z    +0.000, E1   -74.152, E3 +43757.523}
SPL {X  -133.102, Y  +760.274, Z    +0.000, E1   -73.777, E3 +43762.908}
SPL {X  -128.975, Y  +766.169, Z    +0.000, E1   -73.313, E3 +43769.183}
SPL {X  -124.947, Y  +771.425, Z    +0.000, E1   -72.782, E3 +43774.876}
SPL {X  -121.698, Y  +775.357, Z    +0.000, E1   -72.353, E3 +43779.071}
SPL {X  -118.622, Y  +778.858, Z    +0.000, E1   -71.924, E3 +43782.697}
SPL {X   -66.171, Y  +817.165, Z    +0.000, E1   -56.016, E3 +43934.055}
ENDSPLINE

SPLINE
SPL {X  -126.418, Y  +769.557, Z    +0.000, E1   -57.118, E3 +44117.296}
SPL {X  -148.476, Y  +731.097, Z    +0.000, E1   -47.824, E3 +44132.452}
SPL {X  -156.642, Y  +704.059, Z    +0.000, E1   -33.659, E3 +44137.094}
SPL {X  -159.317, Y  +686.157, Z    +0.000, E1   -18.660, E3 +44138.584}
SPL {X  -159.973, Y  +673.799, Z    +0.000, E1    -5.345, E3 +44139.033}
SPL {X  -159.990, Y  +669.500, Z    +0.000, E1    +0.000, E3 +44139.073}
SPL {X  -159.990, Y  +667.794, Z    +0.000, E1    +4.255, E3 +44139.084}
SPL {X  -159.990, Y  +664.091, Z    +0.000, E1   +14.928, E3 +44139.156}
SPL {X  -159.990, Y  +659.599, Z    +0.000, E1   +28.016, E3 +44139.327}
SPL {X  -159.990, Y  +652.711, Z    +0.000, E1   +44.293, E3 +44139.806}
SPL {X  -159.990, Y  +640.730, Z    +0.000, E1   +60.297, E3 +44141.155}
SPL {X  -159.990, Y  +620.478, Z    +0.000, E1   +70.026, E3 +44144.968}
SPL {X  -159.990, Y  +573.021, Z    +0.000, E1   +74.619, E3 +44158.912}
SPL {X  -154.165, Y  +339.724, Z    +0.000, E1   +75.927, E3 +44254.759}
SPL {X  -150.223, Y  +327.456, Z    +0.000, E1   +75.573, E3 +44265.024}
SPL {X  -136.549, Y  +299.126, Z    +0.000, E1   +77.537, E3 +44257.914}
ENDSPLINE

SPLINE
SPL {X  -136.862, Y  +299.641, Z    +0.000, E1   +76.604, E3 +44266.556}
ENDSPLINE

SPLINE
SPL {X  -136.434, Y  +298.938, Z    +0.000, E1   +75.982, E3 +44272.447}
SPL {X  -135.890, Y  +298.057, Z    +0.000, E1   +75.040, E3 +44280.913}
SPL {X  -134.349, Y  +295.626, Z    +0.000, E1   +74.322, E3 +44287.760}
SPL {X  -131.287, Y  +291.064, Z    +0.000, E1   +73.972, E3 +44292.573}
SPL {X  -128.265, Y  +286.871, Z    +0.000, E1   +73.613, E3 +44297.029}
SPL {X  -125.161, Y  +282.843, Z    +0.000, E1   +73.232, E3 +44301.301}
SPL {X  -122.038, Y  +279.042, Z    +0.000, E1   +72.832, E3 +44305.281}
SPL {X  -118.642, Y  +275.165, Z    +0.000, E1   +72.381, E3 +44309.244}
SPL {X   -66.040, Y  +236.776, Z    +0.000, E1   +55.694, E3 +44470.607}
ENDSPLINE

SPLINE
SPL {X  -127.452, Y  +285.790, Z    +0.000, E1   +56.591, E3 +44644.552}
SPL {X  -151.591, Y  +331.344, Z    +0.000, E1   +43.870, E3 +44660.652}
SPL {X  -158.135, Y  +358.205, Z    +0.000, E1   +26.984, E3 +44664.379}
SPL {X  -159.602, Y  +371.361, Z    +0.000, E1   +14.835, E3 +44665.275}
SPL {X  -159.981, Y  +380.818, Z    +0.000, E1    +4.512, E3 +44665.553}
SPL {X  -159.990, Y  +384.681, Z    +0.000, E1    -0.222, E3 +44665.582}
SPL {X  -159.990, Y  +387.626, Z    +0.000, E1    -8.190, E3 +44665.611}
SPL {X  -159.990, Y  +390.340, Z    +0.000, E1   -15.987, E3 +44665.675}
SPL {X  -159.990, Y  +394.216, Z    +0.000, E1   -27.062, E3 +44665.837}
SPL {X  -159.990, Y  +399.855, Z    +0.000, E1   -40.916, E3 +44666.208}
SPL {X  -159.990, Y  +405.475, Z    +0.000, E1   -51.039, E3 +44666.725}
SPL {X  -159.990, Y  +414.231, Z    +0.000, E1   -60.575, E3 +44667.909}
SPL {X  -159.990, Y  +462.953, Z    +0.000, E1   -73.611, E3 +44679.648}
SPL {X  -153.839, Y  +715.436, Z    +0.000, E1   -75.884, E3 +44782.079}
SPL {X  -148.840, Y  +730.182, Z    +0.000, E1   -75.434, E3 +44794.655}
SPL {X  -143.409, Y  +742.426, Z    +0.000, E1   -74.905, E3 +44806.167}
SPL {X  -139.557, Y  +749.735, Z    +0.000, E1   -74.483, E3 +44813.515}
SPL {X  -136.371, Y  +755.165, Z    +0.000, E1   -74.152, E3 +44819.061}
SPL {X  -133.102, Y  +760.274, Z    +0.000, E1   -73.777, E3 +44824.446}
SPL {X  -128.975, Y  +766.169, Z    +0.000, E1   -73.313, E3 +44830.722}
SPL {X  -124.947, Y  +771.425, Z    +0.000, E1   -72.782, E3 +44836.415}
SPL {X  -121.698, Y  +775.357, Z    +0.000, E1   -72.353, E3 +44840.609}
SPL {X  -118.622, Y  +778.858, Z    +0.000, E1   -71.924, E3 +44844.235}
SPL {X   -66.171, Y  +817.165, Z    +0.000, E1   -56.016, E3 +44995.593}
ENDSPLINE

SPLINE
SPL {X  -126.418, Y  +769.557, Z    +0.000, E1   -57.118, E3 +45178.835}
SPL {X  -148.476, Y  +731.097, Z    +0.000, E1   -47.824, E3 +45193.991}
SPL {X  -156.642, Y  +704.059, Z    +0.000, E1   -33.659, E3 +45198.632}
SPL {X  -159.317, Y  +686.157, Z    +0.000, E1   -18.660, E3 +45200.123}
SPL {X  -159.973, Y  +673.799, Z    +0.000, E1    -5.345, E3 +45200.571}
SPL {X  -159.990, Y  +669.500, Z    +0.000, E1    +0.000, E3 +45200.611}
SPL {X  -159.990, Y  +667.794, Z    +0.000, E1    +4.255, E3 +45200.623}
SPL {X  -159.990, Y  +664.091, Z    +0.000, E1   +14.928, E3 +45200.695}
SPL {X  -159.990, Y  +659.599, Z    +0.000, E1   +28.016, E3 +45200.865}
SPL {X  -159.990, Y  +652.711, Z    +0.000, E1   +44.293, E3 +45201.344}
SPL {X  -159.990, Y  +640.730, Z    +0.000, E1   +60.297, E3 +45202.693}
SPL {X  -159.990, Y  +620.478, Z    +0.000, E1   +70.026, E3 +45206.507}
SPL {X  -159.990, Y  +573.021, Z    +0.000, E1   +74.619, E3 +45220.451}
SPL {X  -154.165, Y  +339.724, Z    +0.000, E1   +75.927, E3 +45316.298}
SPL {X  -150.223, Y  +327.456, Z    +0.000, E1   +75.573, E3 +45326.562}
SPL {X  -136.549, Y  +299.126, Z    +0.000, E1   +77.537, E3 +45319.452}
ENDSPLINE

SPLINE
SPL {X  -136.862, Y  +299.641, Z    +0.000, E1   +76.604, E3 +45328.094}
ENDSPLINE

SPLINE
SPL {X  -136.434, Y  +298.938, Z    +0.000, E1   +75.982, E3 +45333.986}
SPL {X  -135.890, Y  +298.057, Z    +0.000, E1   +75.040, E3 +45342.452}
SPL {X  -134.349, Y  +295.626, Z    +0.000, E1   +74.322, E3 +45349.299}
SPL {X  -131.287, Y  +291.064, Z    +0.000, E1   +73.972, E3 +45354.111}
SPL {X  -128.265, Y  +286.871, Z    +0.000, E1   +73.613, E3 +45358.567}
SPL {X  -125.161, Y  +282.843, Z    +0.000, E1   +73.232, E3 +45362.839}
SPL {X  -122.038, Y  +279.042, Z    +0.000, E1   +72.832, E3 +45366.819}
SPL {X  -118.642, Y  +275.165, Z    +0.000, E1   +72.381, E3 +45370.782}
SPL {X   -66.040, Y  +236.776, Z    +0.000, E1   +55.694, E3 +45532.146}
ENDSPLINE

SPLINE
SPL {X  -127.452, Y  +285.790, Z    +0.000, E1   +56.591, E3 +45706.091}
SPL {X  -151.591, Y  +331.344, Z    +0.000, E1   +43.870, E3 +45722.190}
SPL {X  -158.135, Y  +358.205, Z    +0.000, E1   +26.984, E3 +45725.918}
SPL {X  -159.602, Y  +371.361, Z    +0.000, E1   +14.835, E3 +45726.814}
SPL {X  -159.981, Y  +380.818, Z    +0.000, E1    +4.512, E3 +45727.092}
SPL {X  -159.990, Y  +384.681, Z    +0.000, E1    -0.222, E3 +45727.121}
SPL {X  -159.990, Y  +387.626, Z    +0.000, E1    -8.190, E3 +45727.149}
SPL {X  -159.990, Y  +390.340, Z    +0.000, E1   -15.987, E3 +45727.214}
SPL {X  -159.990, Y  +394.216, Z    +0.000, E1   -27.062, E3 +45727.375}
SPL {X  -159.990, Y  +399.855, Z    +0.000, E1   -40.916, E3 +45727.747}
SPL {X  -159.990, Y  +405.475, Z    +0.000, E1   -51.039, E3 +45728.263}
SPL {X  -159.990, Y  +414.231, Z    +0.000, E1   -60.575, E3 +45729.448}
SPL {X  -159.990, Y  +462.953, Z    +0.000, E1   -73.611, E3 +45741.187}
SPL {X  -153.839, Y  +715.436, Z    +0.000, E1   -75.884, E3 +45843.617}
SPL {X  -148.840, Y  +730.182, Z    +0.000, E1   -75.434, E3 +45856.194}
SPL {X  -143.409, Y  +742.426, Z    +0.000, E1   -74.905, E3 +45867.706}
SPL {X  -139.557, Y  +749.735, Z    +0.000, E1   -74.483, E3 +45875.054}
SPL {X  -136.371, Y  +755.165, Z    +0.000, E1   -74.152, E3 +45880.600}
SPL {X  -131.455, Y  +762.694, Z    +0.000, E1   -73.615, E3 +45888.518}
SPL {X  -125.933, Y  +770.180, Z    +0.000, E1   -72.934, E3 +45896.582}
SPL {X  -121.698, Y  +775.357, Z    +0.000, E1   -72.353, E3 +45902.148}
SPL {X  -118.622, Y  +778.858, Z    +0.000, E1   -71.924, E3 +45905.774}
SPL {X   -66.171, Y  +817.165, Z    +0.000, E1   -56.016, E3 +46057.132}
ENDSPLINE

SPLINE
SPL {X  -126.418, Y  +769.557, Z    +0.000, E1   -57.118, E3 +46240.373}
SPL {X  -145.244, Y  +738.589, Z    +0.000, E1   -50.405, E3 +46253.615}
SPL {X  -150.151, Y  +726.741, Z    +0.000, E1   -46.068, E3 +46256.541}
SPL {X  -156.642, Y  +704.059, Z    +0.000, E1   -33.659, E3 +46260.171}
SPL {X  -159.317, Y  +686.157, Z    +0.000, E1   -18.660, E3 +46261.661}
SPL {X  -159.973, Y  +673.799, Z    +0.000, E1    -5.345, E3 +46262.110}
SPL {X  -159.990, Y  +669.500, Z    +0.000, E1    +0.000, E3 +46262.150}
SPL {X  -159.990, Y  +667.794, Z    +0.000, E1    +4.255, E3 +46262.161}
SPL {X  -159.990, Y  +664.091, Z    +0.000, E1   +14.928, E3 +46262.233}
SPL {X  -159.990, Y  +659.599, Z    +0.000, E1   +28.016, E3 +46262.404}
SPL {X  -159.990, Y  +652.711, Z    +0.000, E1   +44.293, E3 +46262.883}
SPL {X  -159.990, Y  +640.730, Z    +0.000, E1   +60.297, E3 +46264.232}
SPL {X  -159.990, Y  +620.478, Z    +0.000, E1   +70.026, E3 +46268.045}
SPL {X  -159.990, Y  +573.021, Z    +0.000, E1   +74.619, E3 +46281.989}
SPL {X  -154.165, Y  +339.724, Z    +0.000, E1   +75.927, E3 +46377.836}
SPL {X  -150.223, Y  +327.456, Z    +0.000, E1   +75.573, E3 +46388.101}
SPL {X  -136.549, Y  +299.126, Z    +0.000, E1   +77.537, E3 +46380.991}
ENDSPLINE

SPLINE
SPL {X  -136.626, Y  +299.252, Z    +0.000, E1   +76.314, E3 +46392.641}
ENDSPLINE

SPLINE
SPL {X  -135.890, Y  +298.057, Z    +0.000, E1   +75.040, E3 +46403.990}
SPL {X  -134.349, Y  +295.626, Z    +0.000, E1   +74.322, E3 +46410.837}
SPL {X  -131.287, Y  +291.064, Z    +0.000, E1   +73.972, E3 +46415.650}
SPL {X  -128.265, Y  +286.871, Z    +0.000, E1   +73.613, E3 +46420.106}
SPL {X  -125.161, Y  +282.843, Z    +0.000, E1   +73.232, E3 +46424.378}
SPL {X  -122.038, Y  +279.042, Z    +0.000, E1   +72.832, E3 +46428.357}
SPL {X  -118.642, Y  +275.165, Z    +0.000, E1   +72.381, E3 +46432.321}
SPL {X   -66.040, Y  +236.776, Z    +0.000, E1   +55.694, E3 +46593.684}
ENDSPLINE

SPLINE
SPL {X  -127.452, Y  +285.790, Z    +0.000, E1   +56.591, E3 +46767.629}
SPL {X  -151.591, Y  +331.344, Z    +0.000, E1   +43.870, E3 +46783.729}
SPL {X  -158.135, Y  +358.205, Z    +0.000, E1   +26.984, E3 +46787.456}
SPL {X  -159.602, Y  +371.361, Z    +0.000, E1   +14.835, E3 +46788.352}
SPL {X  -159.981, Y  +380.818, Z    +0.000, E1    +4.512, E3 +46788.630}
SPL {X  -159.990, Y  +384.681, Z    +0.000, E1    -0.222, E3 +46788.659}
SPL {X  -159.990, Y  +387.626, Z    +0.000, E1    -8.190, E3 +46788.687}
SPL {X  -159.990, Y  +390.340, Z    +0.000, E1   -15.987, E3 +46788.752}
SPL {X  -159.990, Y  +394.216, Z    +0.000, E1   -27.062, E3 +46788.914}
SPL {X  -159.990, Y  +399.855, Z    +0.000, E1   -40.916, E3 +46789.285}
SPL {X  -159.990, Y  +405.475, Z    +0.000, E1   -51.039, E3 +46789.802}
SPL {X  -159.990, Y  +414.231, Z    +0.000, E1   -60.575, E3 +46790.986}
SPL {X  -159.990, Y  +462.953, Z    +0.000, E1   -73.611, E3 +46802.725}
SPL {X  -153.839, Y  +715.436, Z    +0.000, E1   -75.884, E3 +46905.156}
SPL {X  -149.923, Y  +727.355, Z    +0.000, E1   -75.515, E3 +46915.266}
SPL {X  -145.995, Y  +736.939, Z    +0.000, E1   -75.150, E3 +46924.000}
SPL {X  -142.305, Y  +744.618, Z    +0.000, E1   -74.773, E3 +46931.444}
SPL {X  -139.557, Y  +749.735, Z    +0.000, E1   -74.483, E3 +46936.592}
SPL {X  -136.371, Y  +755.165, Z    +0.000, E1   -74.152, E3 +46942.138}
SPL {X  -133.102, Y  +760.274, Z    +0.000, E1   -73.777, E3 +46947.523}
SPL {X  -128.975, Y  +766.169, Z    +0.000, E1   -73.313, E3 +46953.799}
SPL {X  -124.947, Y  +771.425, Z    +0.000, E1   -72.782, E3 +46959.492}
SPL {X  -121.698, Y  +775.357, Z    +0.000, E1   -72.353, E3 +46963.686}
SPL {X  -118.622, Y  +778.858, Z    +0.000, E1   -71.924, E3 +46967.312}
SPL {X   -66.171, Y  +817.165, Z    +0.000, E1   -56.016, E3 +47118.670}
ENDSPLINE

SPLINE
SPL {X  -126.418, Y  +769.557, Z    +0.000, E1   -57.118, E3 +47301.912}
SPL {X  -148.476, Y  +731.097, Z    +0.000, E1   -47.824, E3 +47317.068}
SPL {X  -156.642, Y  +704.059, Z    +0.000, E1   -33.659, E3 +47321.709}
SPL {X  -159.317, Y  +686.157, Z    +0.000, E1   -18.660, E3 +47323.200}
SPL {X  -159.907, Y  +676.666, Z    +0.000, E1    -8.555, E3 +47323.598}
SPL {X  -159.990, Y  +669.586, Z    +0.000, E1    -0.216, E3 +47323.688}
SPL {X  -159.990, Y  +667.794, Z    +0.000, E1    +4.255, E3 +47323.699}
SPL {X  -159.990, Y  +664.091, Z    +0.000, E1   +14.928, E3 +47323.772}
SPL {X  -159.990, Y  +659.599, Z    +0.000, E1   +28.016, E3 +47323.942}
SPL {X  -159.990, Y  +652.711, Z    +0.000, E1   +44.293, E3 +47324.421}
SPL {X  -159.990, Y  +640.730, Z    +0.000, E1   +60.297, E3 +47325.770}
SPL {X  -159.990, Y  +620.478, Z    +0.000, E1   +70.026, E3 +47329.584}
SPL {X  -159.990, Y  +573.021, Z    +0.000, E1   +74.619, E3 +47343.528}
SPL {X  -154.165, Y  +339.724, Z    +0.000, E1   +75.927, E3 +47439.374}
SPL {X  -150.223, Y  +327.456, Z    +0.000, E1   +75.573, E3 +47449.639}
SPL {X  -136.549, Y  +299.126, Z    +0.000, E1   +77.537, E3 +47442.529}
ENDSPLINE

SPLINE
SPL {X  -136.862, Y  +299.641, Z    +0.000, E1   +76.604, E3 +47451.171}
ENDSPLINE

SPLINE
SPL {X  -136.434, Y  +298.938, Z    +0.000, E1   +75.982, E3 +47457.062}
SPL {X  -135.890, Y  +298.057, Z    +0.000, E1   +75.040, E3 +47465.528}
SPL {X  -134.349, Y  +295.626, Z    +0.000, E1   +74.322, E3 +47472.376}
SPL {X  -131.287, Y  +291.064, Z    +0.000, E1   +73.972, E3 +47477.188}
SPL {X  -128.265, Y  +286.871, Z    +0.000, E1   +73.613, E3 +47481.644}
SPL {X  -125.161, Y  +282.843, Z    +0.000, E1   +73.232, E3 +47485.916}
SPL {X  -122.038, Y  +279.042, Z    +0.000, E1   +72.832, E3 +47489.896}
SPL {X  -118.642, Y  +275.165, Z    +0.000, E1   +72.381, E3 +47493.859}
SPL {X   -66.040, Y  +236.776, Z    +0.000, E1   +55.694, E3 +47655.223}
ENDSPLINE

SPLINE
SPL {X  -127.452, Y  +285.790, Z    +0.000, E1   +56.591, E3 +47829.168}
SPL {X  -148.001, Y  +321.733, Z    +0.000, E1   +47.810, E3 +47843.271}
SPL {X  -154.604, Y  +341.337, Z    +0.000, E1   +38.630, E3 +47847.045}
SPL {X  -158.135, Y  +358.205, Z    +0.000, E1   +26.984, E3 +47848.995}
SPL {X  -159.602, Y  +371.361, Z    +0.000, E1   +14.835, E3 +47849.891}
SPL {X  -159.981, Y  +380.818, Z    +0.000, E1    +4.512, E3 +47850.169}
SPL {X  -159.990, Y  +384.681, Z    +0.000, E1    -0.222, E3 +47850.198}
SPL {X  -159.990, Y  +389.079, Z    +0.000, E1   -12.017, E3 +47850.261}
SPL {X  -159.990, Y  +394.216, Z    +0.000, E1   -27.062, E3 +47850.452}
SPL {X  -159.990, Y  +399.855, Z    +0.000, E1   -40.916, E3 +47850.823}
SPL {X  -159.990, Y  +405.475, Z    +0.000, E1   -51.039, E3 +47851.340}
SPL {X  -159.990, Y  +414.231, Z    +0.000, E1   -60.575, E3 +47852.525}
SPL {X  -159.990, Y  +462.953, Z    +0.000, E1   -73.611, E3 +47864.264}
SPL {X  -153.839, Y  +715.436, Z    +0.000, E1   -75.884, E3 +47966.694}
SPL {X  -148.840, Y  +730.182, Z    +0.000, E1   -75.434, E3 +47979.271}
SPL {X  -143.409, Y  +742.426, Z    +0.000, E1   -74.905, E3 +47990.783}
SPL {X  -139.557, Y  +749.735, Z    +0.000, E1   -74.483, E3 +47998.131}
SPL {X  -136.371, Y  +755.165, Z    +0.000, E1   -74.152, E3 +48003.677}
SPL {X  -133.102, Y  +760.274, Z    +0.000, E1   -73.777, E3 +48009.062}
SPL {X  -128.975, Y  +766.169, Z    +0.000, E1   -73.313, E3 +48015.337}
SPL {X  -124.947, Y  +771.425, Z    +0.000, E1   -72.782, E3 +48021.030}
SPL {X  -121.698, Y  +775.357, Z    +0.000, E1   -72.353, E3 +48025.225}
SPL {X  -118.622, Y  +778.858, Z    +0.000, E1   -71.924, E3 +48028.851}
SPL {X   -66.171, Y  +817.165, Z    +0.000, E1   -56.016, E3 +48180.209}
ENDSPLINE

SPLINE
SPL {X  -126.418, Y  +769.557, Z    +0.000, E1   -57.118, E3 +48363.450}
SPL {X  -145.244, Y  +738.589, Z    +0.000, E1   -50.405, E3 +48376.692}
SPL {X  -150.151, Y  +726.741, Z    +0.000, E1   -46.068, E3 +48379.618}
SPL {X  -156.642, Y  +704.059, Z    +0.000, E1   -33.659, E3 +48383.248}
SPL {X  -159.317, Y  +686.157, Z    +0.000, E1   -18.660, E3 +48384.738}
SPL {X  -159.973, Y  +673.799, Z    +0.000, E1    -5.345, E3 +48385.187}
SPL {X  -159.990, Y  +669.500, Z    +0.000, E1    +0.000, E3 +48385.227}
SPL {X  -159.990, Y  +667.794, Z    +0.000, E1    +4.255, E3 +48385.238}
SPL {X  -159.990, Y  +664.091, Z    +0.000, E1   +14.928, E3 +48385.310}
SPL {X  -159.990, Y  +658.301, Z    +0.000, E1   +31.283, E3 +48385.563}
SPL {X  -159.990, Y  +650.845, Z    +0.000, E1   +47.892, E3 +48386.108}
SPL {X  -159.990, Y  +640.730, Z    +0.000, E1   +60.297, E3 +48387.309}
SPL {X  -159.990, Y  +620.478, Z    +0.000, E1   +70.026, E3 +48391.122}
SPL {X  -159.990, Y  +573.021, Z    +0.000, E1   +74.619, E3 +48405.066}
SPL {X  -154.165, Y  +339.724, Z    +0.000, E1   +75.927, E3 +48500.913}
SPL {X  -150.223, Y  +327.456, Z    +0.000, E1   +75.573, E3 +48511.178}
SPL {X  -136.549, Y  +299.126, Z    +0.000, E1   +77.537, E3 +48504.068}
ENDSPLINE

SPLINE
SPL {X  -136.862, Y  +299.641, Z    +0.000, E1   +76.604, E3 +48512.710}
ENDSPLINE

SPLINE
SPL {X  -136.434, Y  +298.938, Z    +0.000, E1   +75.982, E3 +48518.601}
SPL {X  -135.890, Y  +298.057, Z    +0.000, E1   +75.040, E3 +48527.067}
SPL {X  -134.349, Y  +295.626, Z    +0.000, E1   +74.322, E3 +48533.914}
SPL {X  -131.287, Y  +291.064, Z    +0.000, E1   +73.972, E3 +48538.727}
SPL {X  -128.265, Y  +286.871, Z    +0.000, E1   +73.613, E3 +48543.183}
SPL {X  -125.161, Y  +282.843, Z    +0.000, E1   +73.232, E3 +48547.454}
SPL {X  -122.038, Y  +279.042, Z    +0.000, E1   +72.832, E3 +48551.434}
SPL {X  -118.642, Y  +275.165, Z    +0.000, E1   +72.381, E3 +48555.398}
SPL {X   -66.040, Y  +236.776, Z    +0.000, E1   +55.694, E3 +48716.761}
ENDSPLINE

SPLINE
SPL {X  -127.452, Y  +285.790, Z    +0.000, E1   +56.591, E3 +48890.706}
SPL {X  -151.591, Y  +331.344, Z    +0.000, E1   +43.870, E3 +48906.806}
SPL {X  -158.135, Y  +358.205, Z    +0.000, E1   +26.984, E3 +48910.533}
SPL {X  -159.602, Y  +371.361, Z    +0.000, E1   +14.835, E3 +48911.429}
SPL {X  -159.981, Y  +380.818, Z    +0.000, E1    +4.512, E3 +48911.707}
SPL {X  -159.990, Y  +384.681, Z    +0.000, E1    -0.222, E3 +48911.736}
SPL {X  -159.990, Y  +387.626, Z    +0.000, E1    -8.190, E3 +48911.764}
SPL {X  -159.990, Y  +390.340, Z    +0.000, E1   -15.987, E3 +48911.829}
SPL {X  -159.990, Y  +394.216, Z    +0.000, E1   -27.062, E3 +48911.991}
SPL {X  -159.990, Y  +399.855, Z    +0.000, E1   -40.916, E3 +48912.362}
SPL {X  -159.990, Y  +405.475, Z    +0.000, E1   -51.039, E3 +48912.879}
SPL {X  -159.990, Y  +414.231, Z    +0.000, E1   -60.575, E3 +48914.063}
SPL {X  -159.990, Y  +462.953, Z    +0.000, E1   -73.611, E3 +48925.802}
SPL {X  -153.839, Y  +715.436, Z    +0.000, E1   -75.884, E3 +49028.233}
SPL {X  -149.923, Y  +727.355, Z    +0.000, E1   -75.515, E3 +49038.343}
SPL {X  -145.995, Y  +736.939, Z    +0.000, E1   -75.150, E3 +49047.077}
SPL {X  -141.012, Y  +747.080, Z    +0.000, E1   -74.661, E3 +49056.929}
SPL {X  -136.371, Y  +755.165, Z    +0.000, E1   -74.152, E3 +49065.215}
SPL {X  -131.455, Y  +762.694, Z    +0.000, E1   -73.615, E3 +49073.133}
SPL {X  -125.933, Y  +770.180, Z    +0.000, E1   -72.934, E3 +49081.198}
SPL {X  -121.698, Y  +775.357, Z    +0.000, E1   -72.353, E3 +49086.763}
SPL {X  -118.622, Y  +778.858, Z    +0.000, E1   -71.924, E3 +49090.389}
SPL {X   -66.171, Y  +817.165, Z    +0.000, E1   -56.016, E3 +49241.747}
ENDSPLINE

SPLINE
SPL {X  -126.418, Y  +769.557, Z    +0.000, E1   -57.118, E3 +49424.989}
SPL {X  -145.244, Y  +738.589, Z    +0.000, E1   -50.405, E3 +49438.230}
SPL {X  -150.151, Y  +726.741, Z    +0.000, E1   -46.068, E3 +49441.157}
SPL {X  -156.642, Y  +704.059, Z    +0.000, E1   -33.659, E3 +49444.786}
SPL {X  -159.317, Y  +686.157, Z    +0.000, E1   -18.660, E3 +49446.276}
SPL {X  -159.973, Y  +673.799, Z    +0.000, E1    -5.345, E3 +49446.725}
SPL {X  -159.990, Y  +669.500, Z    +0.000, E1    +0.000, E3 +49446.765}
SPL {X  -159.990, Y  +667.794, Z    +0.000, E1    +4.255, E3 +49446.776}
SPL {X  -159.990, Y  +664.091, Z    +0.000, E1   +14.928, E3 +49446.848}
SPL {X  -159.990, Y  +658.301, Z    +0.000, E1   +31.283, E3 +49447.101}
SPL {X  -159.990, Y  +650.845, Z    +0.000, E1   +47.892, E3 +49447.646}
SPL {X  -159.990, Y  +640.730, Z    +0.000, E1   +60.297, E3 +49448.847}
SPL {X  -159.990, Y  +620.478, Z    +0.000, E1   +70.026, E3 +49452.661}
SPL {X  -159.990, Y  +573.021, Z    +0.000, E1   +74.619, E3 +49466.604}
SPL {X  -154.165, Y  +339.724, Z    +0.000, E1   +75.927, E3 +49562.451}
SPL {X  -150.223, Y  +327.456, Z    +0.000, E1   +75.573, E3 +49572.716}
SPL {X  -136.549, Y  +299.126, Z    +0.000, E1   +77.537, E3 +49565.606}
ENDSPLINE

SPLINE
SPL {X  -136.862, Y  +299.641, Z    +0.000, E1   +76.604, E3 +49574.248}
ENDSPLINE

SPLINE
SPL {X  -136.434, Y  +298.938, Z    +0.000, E1   +75.982, E3 +49580.139}
SPL {X  -135.890, Y  +298.057, Z    +0.000, E1   +75.040, E3 +49588.605}
SPL {X  -134.349, Y  +295.626, Z    +0.000, E1   +74.322, E3 +49595.453}
SPL {X  -131.287, Y  +291.064, Z    +0.000, E1   +73.972, E3 +49600.265}
SPL {X  -128.265, Y  +286.871, Z    +0.000, E1   +73.613, E3 +49604.721}
SPL {X  -125.161, Y  +282.843, Z    +0.000, E1   +73.232, E3 +49608.993}
SPL {X  -122.038, Y  +279.042, Z    +0.000, E1   +72.832, E3 +49612.973}
SPL {X  -118.642, Y  +275.165, Z    +0.000, E1   +72.381, E3 +49616.936}
SPL {X   -66.040, Y  +236.776, Z    +0.000, E1   +55.694, E3 +49778.299}
ENDSPLINE

SPLINE
SPL {X  -127.452, Y  +285.790, Z    +0.000, E1   +56.591, E3 +49952.245}
SPL {X  -151.591, Y  +331.344, Z    +0.000, E1   +43.870, E3 +49968.344}
SPL {X  -158.135, Y  +358.205, Z    +0.000, E1   +26.984, E3 +49972.072}
SPL {X  -159.602, Y  +371.361, Z    +0.000, E1   +14.835, E3 +49972.968}
SPL {X  -159.981, Y  +380.818, Z    +0.000, E1    +4.512, E3 +49973.246}
SPL {X  -159.990, Y  +384.681, Z    +0.000, E1    -0.222, E3 +49973.274}
SPL {X  -159.990, Y  +387.626, Z    +0.000, E1    -8.190, E3 +49973.303}
SPL {X  -159.990, Y  +390.340, Z    +0.000, E1   -15.987, E3 +49973.367}
SPL {X  -159.990, Y  +394.216, Z    +0.000, E1   -27.062, E3 +49973.529}
SPL {X  -159.990, Y  +399.855, Z    +0.000, E1   -40.916, E3 +49973.900}
SPL {X  -159.990, Y  +405.475, Z    +0.000, E1   -51.039, E3 +49974.417}
SPL {X  -159.990, Y  +414.231, Z    +0.000, E1   -60.575, E3 +49975.602}
SPL {X  -159.990, Y  +462.953, Z    +0.000, E1   -73.611, E3 +49987.341}
SPL {X  -153.839, Y  +715.436, Z    +0.000, E1   -75.884, E3 +50089.771}
SPL {X  -148.840, Y  +730.182, Z    +0.000, E1   -75.434, E3 +50102.348}
SPL {X  -143.409, Y  +742.426, Z    +0.000, E1   -74.905, E3 +50113.860}
SPL {X  -139.557, Y  +749.735, Z    +0.000, E1   -74.483, E3 +50121.208}
SPL {X  -136.371, Y  +755.165, Z    +0.000, E1   -74.152, E3 +50126.753}
SPL {X  -133.102, Y  +760.274, Z    +0.000, E1   -73.777, E3 +50132.139}
SPL {X  -128.975, Y  +766.169, Z    +0.000, E1   -73.313, E3 +50138.414}
SPL {X  -124.947, Y  +771.425, Z    +0.000, E1   -72.782, E3 +50144.107}
SPL {X  -121.698, Y  +775.357, Z    +0.000, E1   -72.353, E3 +50148.301}
SPL {X  -118.622, Y  +778.858, Z    +0.000, E1   -71.924, E3 +50151.927}
SPL {X   -66.171, Y  +817.165, Z    +0.000, E1   -56.016, E3 +50303.286}
ENDSPLINE

SPLINE
SPL {X  -126.418, Y  +769.557, Z    +0.000, E1   -57.118, E3 +50486.527}
SPL {X  -145.244, Y  +738.589, Z    +0.000, E1   -50.405, E3 +50499.769}
SPL {X  -150.151, Y  +726.741, Z    +0.000, E1   -46.068, E3 +50502.695}
SPL {X  -156.642, Y  +704.059, Z    +0.000, E1   -33.659, E3 +50506.325}
SPL {X  -159.317, Y  +686.157, Z    +0.000, E1   -18.660, E3 +50507.815}
SPL {X  -159.973, Y  +673.799, Z    +0.000, E1    -5.345, E3 +50508.264}
SPL {X  -159.990, Y  +669.500, Z    +0.000, E1    +0.000, E3 +50508.304}
SPL {X  -159.990, Y  +667.794, Z    +0.000, E1    +4.255, E3 +50508.315}
SPL {X  -159.990, Y  +664.091, Z    +0.000, E1   +14.928, E3 +50508.387}
SPL {X  -159.990, Y  +659.599, Z    +0.000, E1   +28.016, E3 +50508.557}
SPL {X  -159.990, Y  +652.711, Z    +0.000, E1   +44.293, E3 +50509.037}
SPL {X  -159.990, Y  +640.730, Z    +0.000, E1   +60.297, E3 +50510.386}
SPL {X  -159.990, Y  +620.478, Z    +0.000, E1   +70.026, E3 +50514.199}
SPL {X  -159.990, Y  +573.021, Z    +0.000, E1   +74.619, E3 +50528.143}
SPL {X  -154.165, Y  +339.724, Z    +0.000, E1   +75.927, E3 +50623.990}
SPL {X  -150.571, Y  +328.416, Z    +0.000, E1   +75.599, E3 +50633.435}
SPL {X  -148.206, Y  +322.236, Z    +0.000, E1   +75.365, E3 +50638.979}
SPL {X  -136.549, Y  +299.126, Z    +0.000, E1   +77.537, E3 +50627.145}
ENDSPLINE

SPLINE
SPL {X  -136.862, Y  +299.641, Z    +0.000, E1   +76.604, E3 +50635.787}
ENDSPLINE

SPLINE
SPL {X  -136.434, Y  +298.938, Z    +0.000, E1   +75.982, E3 +50641.678}
SPL {X  -135.890, Y  +298.057, Z    +0.000, E1   +75.040, E3 +50650.144}
SPL {X  -134.349, Y  +295.626, Z    +0.000, E1   +74.322, E3 +50656.991}
SPL {X  -131.287, Y  +291.064, Z    +0.000, E1   +73.972, E3 +50661.804}
SPL {X  -128.265, Y  +286.871, Z    +0.000, E1   +73.613, E3 +50666.260}
SPL {X  -125.161, Y  +282.843, Z    +0.000, E1   +73.232, E3 +50670.531}
SPL {X  -122.038, Y  +279.042, Z    +0.000, E1   +72.832, E3 +50674.511}
SPL {X  -118.642, Y  +275.165, Z    +0.000, E1   +72.381, E3 +50678.474}
SPL {X   -66.040, Y  +236.776, Z    +0.000, E1   +55.694, E3 +50839.838}
ENDSPLINE

SPLINE
SPL {X  -127.452, Y  +285.790, Z    +0.000, E1   +56.591, E3 +51013.783}
SPL {X  -151.591, Y  +331.344, Z    +0.000, E1   +43.870, E3 +51029.883}
SPL {X  -158.135, Y  +358.205, Z    +0.000, E1   +26.984, E3 +51033.610}
SPL {X  -159.602, Y  +371.361, Z    +0.000, E1   +14.835, E3 +51034.506}
SPL {X  -159.981, Y  +380.818, Z    +0.000, E1    +4.512, E3 +51034.784}
SPL {X  -159.990, Y  +384.681, Z    +0.000, E1    -0.222, E3 +51034.813}
SPL {X  -159.990, Y  +387.626, Z    +0.000, E1    -8.190, E3 +51034.841}
SPL {X  -159.990, Y  +390.340, Z    +0.000, E1   -15.987, E3 +51034.906}
SPL {X  -159.990, Y  +394.216, Z    +0.000, E1   -27.062, E3 +51035.068}
SPL {X  -159.990, Y  +399.855, Z    +0.000, E1   -40.916, E3 +51035.439}
SPL {X  -159.990, Y  +405.475, Z    +0.000, E1   -51.039, E3 +51035.956}
SPL {X  -159.990, Y  +414.231, Z    +0.000, E1   -60.575, E3 +51037.140}
SPL {X  -159.990, Y  +462.953, Z    +0.000, E1   -73.611, E3 +51048.879}
SPL {X  -153.839, Y  +715.436, Z    +0.000, E1   -75.884, E3 +51151.310}
SPL {X  -148.840, Y  +730.182, Z    +0.000, E1   -75.434, E3 +51163.886}
SPL {X  -143.409, Y  +742.426, Z    +0.000, E1   -74.905, E3 +51175.398}
SPL {X  -139.557, Y  +749.735, Z    +0.000, E1   -74.483, E3 +51182.746}
SPL {X  -136.371, Y  +755.165, Z    +0.000, E1   -74.152, E3 +51188.292}
SPL {X  -133.102, Y  +760.274, Z    +0.000, E1   -73.777, E3 +51193.677}
SPL {X  -128.975, Y  +766.169, Z    +0.000, E1   -73.313, E3 +51199.952}
SPL {X  -124.947, Y  +771.425, Z    +0.000, E1   -72.782, E3 +51205.645}
SPL {X  -121.698, Y  +775.357, Z    +0.000, E1   -72.353, E3 +51209.840}
SPL {X  -118.622, Y  +778.858, Z    +0.000, E1   -71.924, E3 +51213.466}
SPL {X   -66.171, Y  +817.165, Z    +0.000, E1   -56.016, E3 +51364.824}
ENDSPLINE

SPLINE
SPL {X  -126.418, Y  +769.557, Z    +0.000, E1   -57.118, E3 +51548.065}
SPL {X  -148.476, Y  +731.097, Z    +0.000, E1   -47.824, E3 +51563.221}
SPL {X  -156.642, Y  +704.059, Z    +0.000, E1   -33.659, E3 +51567.863}
SPL {X  -159.317, Y  +686.157, Z    +0.000, E1   -18.660, E3 +51569.353}
SPL {X  -159.973, Y  +673.799, Z    +0.000, E1    -5.345, E3 +51569.802}
SPL {X  -159.990, Y  +669.500, Z    +0.000, E1    +0.000, E3 +51569.842}
SPL {X  -159.990, Y  +667.794, Z    +0.000, E1    +4.255, E3 +51569.853}
SPL {X  -159.990, Y  +664.091, Z    +0.000, E1   +14.928, E3 +51569.925}
SPL {X  -159.990, Y  +659.599, Z    +0.000, E1   +28.016, E3 +51570.096}
SPL {X  -159.990, Y  +652.711, Z    +0.000, E1   +44.293, E3 +51570.575}
SPL {X  -159.990, Y  +640.730, Z    +0.000, E1   +60.297, E3 +51571.924}
SPL {X  -159.990, Y  +620.478, Z    +0.000, E1   +70.026, E3 +51575.738}
SPL {X  -159.990, Y  +573.021, Z    +0.000, E1   +74.619, E3 +51589.681}
SPL {X  -154.165, Y  +339.724, Z    +0.000, E1   +75.927, E3 +51685.528}
SPL {X  -150.223, Y  +327.456, Z    +0.000, E1   +75.573, E3 +51695.793}
SPL {X  -136.549, Y  +299.126, Z    +0.000, E1   +77.537, E3 +51688.683}
ENDSPLINE

SPLINE
SPL {X  -136.862, Y  +299.641, Z    +0.000, E1   +76.604, E3 +51697.325}
ENDSPLINE

SPLINE
SPL {X  -136.434, Y  +298.938, Z    +0.000, E1   +75.982, E3 +51703.216}
SPL {X  -135.890, Y  +298.057, Z    +0.000, E1   +75.040, E3 +51711.682}
SPL {X  -134.349, Y  +295.626, Z    +0.000, E1   +74.322, E3 +51718.530}
SPL {X  -131.287, Y  +291.064, Z    +0.000, E1   +73.972, E3 +51723.342}
SPL {X  -128.265, Y  +286.871, Z    +0.000, E1   +73.613, E3 +51727.798}
SPL {X  -125.161, Y  +282.843, Z    +0.000, E1   +73.232, E3 +51732.070}
SPL {X  -122.038, Y  +279.042, Z    +0.000, E1   +72.832, E3 +51736.050}
SPL {X  -118.642, Y  +275.165, Z    +0.000, E1   +72.381, E3 +51740.013}
SPL {X   -66.040, Y  +236.776, Z    +0.000, E1   +55.694, E3 +51901.376}
ENDSPLINE

SPLINE
SPL {X  -127.452, Y  +285.790, Z    +0.000, E1   +56.591, E3 +52075.322}
SPL {X  -151.591, Y  +331.344, Z    +0.000, E1   +43.870, E3 +52091.421}
SPL {X  -158.135, Y  +358.205, Z    +0.000, E1   +26.984, E3 +52095.149}
SPL {X  -159.602, Y  +371.361, Z    +0.000, E1   +14.835, E3 +52096.045}
SPL {X  -159.981, Y  +380.818, Z    +0.000, E1    +4.512, E3 +52096.322}
SPL {X  -159.990, Y  +384.681, Z    +0.000, E1    -0.222, E3 +52096.351}
SPL {X  -159.990, Y  +387.626, Z    +0.000, E1    -8.190, E3 +52096.380}
SPL {X  -159.990, Y  +390.340, Z    +0.000, E1   -15.987, E3 +52096.444}
SPL {X  -159.990, Y  +394.216, Z    +0.000, E1   -27.062, E3 +52096.606}
SPL {X  -159.990, Y  +399.855, Z    +0.000, E1   -40.916, E3 +52096.977}
SPL {X  -159.990, Y  +405.475, Z    +0.000, E1   -51.039, E3 +52097.494}
SPL {X  -159.990, Y  +414.231, Z    +0.000, E1   -60.575, E3 +52098.678}
SPL {X  -159.990, Y  +462.953, Z    +0.000, E1   -73.611, E3 +52110.417}
SPL {X  -153.839, Y  +715.436, Z    +0.000, E1   -75.884, E3 +52212.848}
SPL {X  -149.923, Y  +727.355, Z    +0.000, E1   -75.515, E3 +52222.958}
SPL {X  -145.995, Y  +736.939, Z    +0.000, E1   -75.150, E3 +52231.693}
SPL {X  -141.012, Y  +747.080, Z    +0.000, E1   -74.661, E3 +52241.545}
SPL {X  -136.371, Y  +755.165, Z    +0.000, E1   -74.152, E3 +52249.830}
SPL {X  -131.455, Y  +762.694, Z    +0.000, E1   -73.615, E3 +52257.748}
SPL {X  -125.933, Y  +770.180, Z    +0.000, E1   -72.934, E3 +52265.813}
SPL {X  -121.698, Y  +775.357, Z    +0.000, E1   -72.353, E3 +52271.378}
SPL {X  -118.622, Y  +778.858, Z    +0.000, E1   -71.924, E3 +52275.004}
SPL {X   -66.171, Y  +817.165, Z    +0.000, E1   -56.016, E3 +52426.363}
ENDSPLINE

SPLINE
SPL {X  -126.418, Y  +769.557, Z    +0.000, E1   -57.118, E3 +52609.604}
SPL {X  -148.476, Y  +731.097, Z    +0.000, E1   -47.824, E3 +52624.760}
SPL {X  -156.642, Y  +704.059, Z    +0.000, E1   -33.659, E3 +52629.402}
SPL {X  -159.317, Y  +686.157, Z    +0.000, E1   -18.660, E3 +52630.892}
SPL {X  -159.907, Y  +676.666, Z    +0.000, E1    -8.555, E3 +52631.290}
SPL {X  -159.990, Y  +669.586, Z    +0.000, E1    -0.216, E3 +52631.380}
SPL {X  -159.990, Y  +667.794, Z    +0.000, E1    +4.255, E3 +52631.392}
SPL {X  -159.990, Y  +664.091, Z    +0.000, E1   +14.928, E3 +52631.464}
SPL {X  -159.990, Y  +658.301, Z    +0.000, E1   +31.283, E3 +52631.716}
SPL {X  -159.990, Y  +650.845, Z    +0.000, E1   +47.892, E3 +52632.262}
SPL {X  -159.990, Y  +640.730, Z    +0.000, E1   +60.297, E3 +52633.463}
SPL {X  -159.990, Y  +620.478, Z    +0.000, E1   +70.026, E3 +52637.276}
SPL {X  -159.990, Y  +573.021, Z    +0.000, E1   +74.619, E3 +52651.220}
SPL {X  -154.165, Y  +339.724, Z    +0.000, E1   +75.927, E3 +52747.067}
SPL {X  -150.571, Y  +328.416, Z    +0.000, E1   +75.599, E3 +52756.512}
SPL {X  -148.206, Y  +322.236, Z    +0.000, E1   +75.365, E3 +52762.056}
SPL {X  -136.549, Y  +299.126, Z    +0.000, E1   +77.537, E3 +52750.222}
ENDSPLINE

SPLINE
SPL {X  -136.626, Y  +299.252, Z    +0.000, E1   +76.314, E3 +52761.872}
ENDSPLINE

SPLINE
SPL {X  -135.890, Y  +298.057, Z    +0.000, E1   +75.040, E3 +52773.221}
SPL {X  -134.349, Y  +295.626, Z    +0.000, E1   +74.322, E3 +52780.068}
SPL {X  -131.287, Y  +291.064, Z    +0.000, E1   +73.972, E3 +52784.881}
SPL {X  -128.265, Y  +286.871, Z    +0.000, E1   +73.613, E3 +52789.337}
SPL {X  -125.161, Y  +282.843, Z    +0.000, E1   +73.232, E3 +52793.608}
SPL {X  -122.038, Y  +279.042, Z    +0.000, E1   +72.832, E3 +52797.588}
SPL {X  -118.642, Y  +275.165, Z    +0.000, E1   +72.381, E3 +52801.551}
SPL {X   -66.040, Y  +236.776, Z    +0.000, E1   +55.694, E3 +52962.915}
ENDSPLINE

SPLINE
SPL {X  -127.452, Y  +285.790, Z    +0.000, E1   +56.591, E3 +53136.860}
SPL {X  -151.591, Y  +331.344, Z    +0.000, E1   +43.870, E3 +53152.959}
SPL {X  -158.135, Y  +358.205, Z    +0.000, E1   +26.984, E3 +53156.687}
SPL {X  -159.602, Y  +371.361, Z    +0.000, E1   +14.835, E3 +53157.583}
SPL {X  -159.981, Y  +380.818, Z    +0.000, E1    +4.512, E3 +53157.861}
SPL {X  -159.990, Y  +384.681, Z    +0.000, E1    -0.222, E3 +53157.890}
SPL {X  -159.990, Y  +387.626, Z    +0.000, E1    -8.190, E3 +53157.918}
SPL {X  -159.990, Y  +390.340, Z    +0.000, E1   -15.987, E3 +53157.983}
SPL {X  -159.990, Y  +394.216, Z    +0.000, E1   -27.062, E3 +53158.145}
SPL {X  -159.990, Y  +399.855, Z    +0.000, E1   -40.916, E3 +53158.516}
SPL {X  -159.990, Y  +405.475, Z    +0.000, E1   -51.039, E3 +53159.033}
SPL {X  -159.990, Y  +414.231, Z    +0.000, E1   -60.575, E3 +53160.217}
SPL {X  -159.990, Y  +462.953, Z    +0.000, E1   -73.611, E3 +53171.956}
SPL {X  -153.839, Y  +715.436, Z    +0.000, E1   -75.884, E3 +53274.386}
SPL {X  -149.923, Y  +727.355, Z    +0.000, E1   -75.515, E3 +53284.496}
SPL {X  -145.995, Y  +736.939, Z    +0.000, E1   -75.150, E3 +53293.231}
SPL {X  -141.012, Y  +747.080, Z    +0.000, E1   -74.661, E3 +53303.083}
SPL {X  -136.371, Y  +755.165, Z    +0.000, E1   -74.152, E3 +53311.369}
SPL {X  -131.455, Y  +762.694, Z    +0.000, E1   -73.615, E3 +53319.287}
SPL {X  -125.933, Y  +770.180, Z    +0.000, E1   -72.934, E3 +53327.352}
SPL {X  -121.698, Y  +775.357, Z    +0.000, E1   -72.353, E3 +53332.917}
SPL {X  -118.622, Y  +778.858, Z    +0.000, E1   -71.924, E3 +53336.543}
SPL {X   -66.171, Y  +817.165, Z    +0.000, E1   -56.016, E3 +53487.901}
ENDSPLINE

SPLINE
SPL {X  -126.418, Y  +769.557, Z    +0.000, E1   -57.118, E3 +53671.142}
SPL {X  -148.476, Y  +731.097, Z    +0.000, E1   -47.824, E3 +53686.298}
SPL {X  -156.642, Y  +704.059, Z    +0.000, E1   -33.659, E3 +53690.940}
SPL {X  -159.317, Y  +686.157, Z    +0.000, E1   -18.660, E3 +53692.430}
SPL {X  -159.973, Y  +673.799, Z    +0.000, E1    -5.345, E3 +53692.879}
SPL {X  -159.990, Y  +669.500, Z    +0.000, E1    +0.000, E3 +53692.919}
SPL {X  -159.990, Y  +667.794, Z    +0.000, E1    +4.255, E3 +53692.930}
SPL {X  -159.990, Y  +664.091, Z    +0.000, E1   +14.928, E3 +53693.002}
SPL {X  -159.990, Y  +659.599, Z    +0.000, E1   +28.016, E3 +53693.173}
SPL {X  -159.990, Y  +652.711, Z    +0.000, E1   +44.293, E3 +53693.652}
SPL {X  -159.990, Y  +640.730, Z    +0.000, E1   +60.297, E3 +53695.001}
SPL {X  -159.990, Y  +620.478, Z    +0.000, E1   +70.026, E3 +53698.814}
SPL {X  -159.990, Y  +573.021, Z    +0.000, E1   +74.619, E3 +53712.758}
SPL {X  -154.165, Y  +339.724, Z    +0.000, E1   +75.927, E3 +53808.605}
SPL {X  -150.223, Y  +327.456, Z    +0.000, E1   +75.573, E3 +53818.870}
SPL {X  -136.549, Y  +299.126, Z    +0.000, E1   +77.537, E3 +53811.760}
ENDSPLINE

SPLINE
SPL {X  -136.862, Y  +299.641, Z    +0.000, E1   +76.604, E3 +53820.402}
ENDSPLINE

SPLINE
SPL {X  -136.434, Y  +298.938, Z    +0.000, E1   +75.982, E3 +53826.293}
SPL {X  -135.890, Y  +298.057, Z    +0.000, E1   +75.040, E3 +53834.759}
SPL {X  -134.349, Y  +295.626, Z    +0.000, E1   +74.322, E3 +53841.606}
SPL {X  -131.287, Y  +291.064, Z    +0.000, E1   +73.972, E3 +53846.419}
SPL {X  -128.265, Y  +286.871, Z    +0.000, E1   +73.613, E3 +53850.875}
SPL {X  -125.161, Y  +282.843, Z    +0.000, E1   +73.232, E3 +53855.147}
SPL {X  -122.038, Y  +279.042, Z    +0.000, E1   +72.832, E3 +53859.127}
SPL {X  -119.499, Y  +276.120, Z    +0.000, E1   +72.482, E3 +53862.146}
SPL {X  -117.726, Y  +274.160, Z    +0.000, E1   +72.234, E3 +53864.109}
SPL {X   -66.040, Y  +236.776, Z    +0.000, E1   +55.694, E3 +54024.453}
ENDSPLINE

SPLINE
SPL {X  -127.452, Y  +285.790, Z    +0.000, E1   +56.591, E3 +54198.399}
SPL {X  -148.001, Y  +321.733, Z    +0.000, E1   +47.810, E3 +54212.502}
SPL {X  -154.604, Y  +341.337, Z    +0.000, E1   +38.630, E3 +54216.276}
SPL {X  -158.135, Y  +358.205, Z    +0.000, E1   +26.984, E3 +54218.226}
SPL {X  -159.602, Y  +371.361, Z    +0.000, E1   +14.835, E3 +54219.122}
SPL {X  -159.981, Y  +380.818, Z    +0.000, E1    +4.512, E3 +54219.399}
SPL {X  -159.990, Y  +384.681, Z    +0.000, E1    -0.222, E3 +54219.428}
SPL {X  -159.990, Y  +387.626, Z    +0.000, E1    -8.190, E3 +54219.457}
SPL {X  -159.990, Y  +390.340, Z    +0.000, E1   -15.987, E3 +54219.521}
SPL {X  -159.990, Y  +394.216, Z    +0.000, E1   -27.062, E3 +54219.683}
SPL {X  -159.990, Y  +399.855, Z    +0.000, E1   -40.916, E3 +54220.054}
SPL {X  -159.990, Y  +405.475, Z    +0.000, E1   -51.039, E3 +54220.571}
SPL {X  -159.990, Y  +414.231, Z    +0.000, E1   -60.575, E3 +54221.755}
SPL {X  -159.990, Y  +462.953, Z    +0.000, E1   -73.611, E3 +54233.494}
SPL {X  -153.839, Y  +715.436, Z    +0.000, E1   -75.884, E3 +54335.925}
SPL {X  -148.840, Y  +730.182, Z    +0.000, E1   -75.434, E3 +54348.502}
SPL {X  -143.409, Y  +742.426, Z    +0.000, E1   -74.905, E3 +54360.014}
SPL {X  -139.557, Y  +749.735, Z    +0.000, E1   -74.483, E3 +54367.362}
SPL {X  -136.371, Y  +755.165, Z    +0.000, E1   -74.152, E3 +54372.907}
SPL {X  -131.455, Y  +762.694, Z    +0.000, E1   -73.615, E3 +54380.825}
SPL {X  -125.933, Y  +770.180, Z    +0.000, E1   -72.934, E3 +54388.890}
SPL {X  -121.698, Y  +775.357, Z    +0.000, E1   -72.353, E3 +54394.455}
SPL {X  -118.622, Y  +778.858, Z    +0.000, E1   -71.924, E3 +54398.081}
SPL {X   -66.171, Y  +817.165, Z    +0.000, E1   -56.016, E3 +54549.440}
ENDSPLINE

SPLINE
SPL {X  -126.418, Y  +769.557, Z    +0.000, E1   -57.118, E3 +54732.681}
SPL {X  -145.244, Y  +738.589, Z    +0.000, E1   -50.405, E3 +54745.922}
SPL {X  -150.151, Y  +726.741, Z    +0.000, E1   -46.068, E3 +54748.849}
SPL {X  -156.642, Y  +704.059, Z    +0.000, E1   -33.659, E3 +54752.479}
SPL {X  -159.317, Y  +686.157, Z    +0.000, E1   -18.660, E3 +54753.969}
SPL {X  -159.973, Y  +673.799, Z    +0.000, E1    -5.345, E3 +54754.417}
SPL {X  -159.990, Y  +669.500, Z    +0.000, E1    +0.000, E3 +54754.457}
SPL {X  -159.990, Y  +667.794, Z    +0.000, E1    +4.255, E3 +54754.469}
SPL {X  -159.990, Y  +664.091, Z    +0.000, E1   +14.928, E3 +54754.541}
SPL {X  -159.990, Y  +659.599, Z    +0.000, E1   +28.016, E3 +54754.711}
SPL {X  -159.990, Y  +652.711, Z    +0.000, E1   +44.293, E3 +54755.191}
SPL {X  -159.990, Y  +640.730, Z    +0.000, E1   +60.297, E3 +54756.540}
SPL {X  -159.990, Y  +620.478, Z    +0.000, E1   +70.026, E3 +54760.353}
SPL {X  -159.990, Y  +573.021, Z    +0.000, E1   +74.619, E3 +54774.297}
SPL {X  -154.165, Y  +339.724, Z    +0.000, E1   +75.927, E3 +54870.144}
SPL {X  -150.571, Y  +328.416, Z    +0.000, E1   +75.599, E3 +54879.589}
SPL {X  -148.206, Y  +322.236, Z    +0.000, E1   +75.365, E3 +54885.133}
SPL {X  -136.549, Y  +299.126, Z    +0.000, E1   +77.537, E3 +54873.299}
ENDSPLINE

SPLINE
SPL {X  -136.862, Y  +299.641, Z    +0.000, E1   +76.604, E3 +54881.941}
ENDSPLINE

SPLINE
SPL {X  -136.434, Y  +298.938, Z    +0.000, E1   +75.982, E3 +54887.832}
SPL {X  -135.890, Y  +298.057, Z    +0.000, E1   +75.040, E3 +54896.298}
SPL {X  -134.349, Y  +295.626, Z    +0.000, E1   +74.322, E3 +54903.145}
SPL {X  -131.287, Y  +291.064, Z    +0.000, E1   +73.972, E3 +54907.957}
SPL {X  -128.265, Y  +286.871, Z    +0.000, E1   +73.613, E3 +54912.413}
SPL {X  -125.161, Y  +282.843, Z    +0.000, E1   +73.232, E3 +54916.685}
SPL {X  -122.038, Y  +279.042, Z    +0.000, E1   +72.832, E3 +54920.665}
SPL {X  -118.642, Y  +275.165, Z    +0.000, E1   +72.381, E3 +54924.628}
SPL {X   -66.040, Y  +236.776, Z    +0.000, E1   +55.694, E3 +55085.992}
ENDSPLINE

SPLINE
SPL {X  -127.452, Y  +285.790, Z    +0.000, E1   +56.591, E3 +55259.937}
SPL {X  -151.591, Y  +331.344, Z    +0.000, E1   +43.870, E3 +55276.036}
SPL {X  -158.135, Y  +358.205, Z    +0.000, E1   +26.984, E3 +55279.764}
SPL {X  -159.602, Y  +371.361, Z    +0.000, E1   +14.835, E3 +55280.660}
SPL {X  -159.981, Y  +380.818, Z    +0.000, E1    +4.512, E3 +55280.938}
SPL {X  -159.990, Y  +384.681, Z    +0.000, E1    -0.222, E3 +55280.967}
SPL {X  -159.990, Y  +387.626, Z    +0.000, E1    -8.190, E3 +55280.995}
SPL {X  -159.990, Y  +390.340, Z    +0.000, E1   -15.987, E3 +55281.060}
SPL {X  -159.990, Y  +394.216, Z    +0.000, E1   -27.062, E3 +55281.222}
SPL {X  -159.990, Y  +399.855, Z    +0.000, E1   -40.916, E3 +55281.593}
SPL {X  -159.990, Y  +405.475, Z    +0.000, E1   -51.039, E3 +55282.110}
SPL {X  -159.990, Y  +414.231, Z    +0.000, E1   -60.575, E3 +55283.294}
SPL {X  -159.990, Y  +462.953, Z    +0.000, E1   -73.611, E3 +55295.033}
SPL {X  -153.839, Y  +715.436, Z    +0.000, E1   -75.884, E3 +55397.463}
SPL {X  -148.840, Y  +730.182, Z    +0.000, E1   -75.434, E3 +55410.040}
SPL {X  -143.409, Y  +742.426, Z    +0.000, E1   -74.905, E3 +55421.552}
SPL {X  -139.557, Y  +749.735, Z    +0.000, E1   -74.483, E3 +55428.900}
SPL {X  -136.371, Y  +755.165, Z    +0.000, E1   -74.152, E3 +55434.446}
SPL {X  -133.102, Y  +760.274, Z    +0.000, E1   -73.777, E3 +55439.831}
SPL {X  -128.975, Y  +766.169, Z    +0.000, E1   -73.313, E3 +55446.106}
SPL {X  -124.947, Y  +771.425, Z    +0.000, E1   -72.782, E3 +55451.799}
SPL {X  -121.698, Y  +775.357, Z    +0.000, E1   -72.353, E3 +55455.994}
SPL {X  -118.622, Y  +778.858, Z    +0.000, E1   -71.924, E3 +55459.620}
SPL {X   -66.171, Y  +817.165, Z    +0.000, E1   -56.016, E3 +55610.978}
ENDSPLINE

